LIN {X 0,Y 220.279,Z 449.432,A -85,B 0,C 180,E1 -22179.651,E2 -22179.651} C_VEL
LIN {X 0,Y 223.173,Z 455.881,A -85,B 0,C 180,E1 -22180.694,E2 -22180.694} C_VEL
LIN {X 0,Y 220.537,Z 499.361,A -85,B 0,C 180,E1 -22182.042,E2 -22182.042} C_VEL
LIN {X 0,Y 218.945,Z 512.319,A -85,B 0,C 180,E1 -22182.756,E2 -22182.756} C_VEL
LIN {X 0,Y 216.728,Z 525.067,A -85,B 0,C 180,E1 -22183.822,E2 -22183.822} C_VEL
LIN {X 0,Y 213.871,Z 536.29,A -85,B 0,C 180,E1 -22185.05,E2 -22185.05} C_VEL
LIN {X 0,Y 210.428,Z 547.967,A -85,B 0,C 180,E1 -22186.792,E2 -22186.792} C_VEL
LIN {X 0,Y 207.087,Z 557.88,A -85,B 0,C 180,E1 -22188.721,E2 -22188.721} C_VEL
LIN {X 0,Y 203.422,Z 566.935,A -85,B 0,C 180,E1 -22190.913,E2 -22190.913} C_VEL
LIN {X 0,Y 199.206,Z 576.115,A -85,B 0,C 180,E1 -22193.787,E2 -22193.787} C_VEL
LIN {X 0,Y 195.527,Z 583.431,A -85,B 0,C 180,E1 -22196.761,E2 -22196.761} C_VEL
LIN {X 0,Y 192.781,Z 588.357,A -85,B 0,C 180,E1 -22199.312,E2 -22199.312} C_VEL
LIN {X 0,Y 189.682,Z 593.549,A -85,B 0,C 180,E1 -22202.779,E2 -22202.779} C_VEL
LIN {X 0,Y 187.622,Z 596.712,A -85,B 0,C 180,E1 -22205.668,E2 -22205.668} C_VEL
LIN {X 0,Y 186.374,Z 598.548,A -85,B 0,C 180,E1 -22207.847,E2 -22207.847} C_VEL
LIN {X 0,Y 184.61,Z 600.806,A -85,B 0,C 180,E1 -22212.13,E2 -22212.13} C_VEL
LIN {X 0,Y 183.947,Z 601.411,A -85,B 0,C 180,E1 -22214.488,E2 -22214.488} C_VEL
LIN {X 0,Y 183.461,Z 601.557,A -85,B 0,C 180,E1 -22216.712,E2 -22216.712} C_VEL
LIN {X 0,Y 183.165,Z 600.608,A -85,B 0,C 180,E1 -22221.172,E2 -22221.172} C_VEL
LIN {X 0,Y 183.462,Z 598.591,A -85,B 0,C 180,E1 -22224.883,E2 -22224.883} C_VEL
LIN {X 0,Y 183.934,Z 595.067,A -85,B 0,C 180,E1 -22228.905,E2 -22228.905} C_VEL
LIN {X 0,Y 184.847,Z 591.015,A -85,B 0,C 180,E1 -22232.179,E2 -22232.179} C_VEL
LIN {X 0,Y 186.289,Z 584.814,A -85,B 0,C 180,E1 -22235.955,E2 -22235.955} C_VEL
LIN {X 0,Y 188.121,Z 578.059,A -85,B 0,C 180,E1 -22239.136,E2 -22239.136} C_VEL
LIN {X 0,Y 190.373,Z 569.662,A -85,B 0,C 180,E1 -22242.255,E2 -22242.255} C_VEL
LIN {X 0,Y 192.597,Z 561.018,A -85,B 0,C 180,E1 -22244.799,E2 -22244.799} C_VEL
LIN {X 0,Y 195.203,Z 550.369,A -85,B 0,C 180,E1 -22247.279,E2 -22247.279} C_VEL
LIN {X 0,Y 197.473,Z 539.775,A -85,B 0,C 180,E1 -22249.22,E2 -22249.22} C_VEL
LIN {X 0,Y 199.436,Z 527.973,A -85,B 0,C 180,E1 -22250.903,E2 -22250.903} C_VEL
LIN {X 0,Y 201.153,Z 515.679,A -85,B 0,C 180,E1 -22252.195,E2 -22252.195} C_VEL
LIN {X 0,Y 202.366,Z 502.967,A -85,B 0,C 180,E1 -22253.14,E2 -22253.14} C_VEL
LIN {X 0,Y 203.145,Z 489.487,A -85,B 0,C 180,E1 -22253.729,E2 -22253.729} C_VEL
LIN {X 0,Y 205.349,Z 437.648,A -85,B 0,C 180,E1 -22255.442,E2 -22255.442} C_VEL
LIN {X 0,Y 202.251,Z 429.977,A -85,B 0,C 180,E1 -22256.283,E2 -22256.283} C_VEL
LIN {X 0,Y 193.557,Z 412.703,A -85,B 0,C 180,E1 -22258.641,E2 -22258.641} C_VEL
LIN {X 0,Y 187.249,Z 402.11,A -85,B 0,C 180,E1 -22260.443,E2 -22260.443} C_VEL
LIN {X 0,Y 185.803,Z 399.476,A -85,B 0,C 180,E1 -22260.889,E2 -22260.889} C_VEL
LIN {X 0,Y 185.553,Z 398.371,A -85,B 0,C 180,E1 -22261.052,E2 -22261.052} C_VEL
LIN {X 0,Y 185.501,Z 398.377,A -85,B 0,C 180,E1 -22264.631,E2 -22264.631} C_VEL
LIN {X 0,Y 185.507,Z 398.376,A -85,B 0,C 180,E1 -22267.312,E2 -22267.312} C_VEL
LIN {X 0,Y 185.497,Z 398.375,A -85,B 0,C 180,E1 -22272.997,E2 -22272.997} C_VEL
LIN {X 0,Y 185.554,Z 398.352,A -85,B 0,C 180,E1 -22277.017,E2 -22277.017} C_VEL
LIN {X 0,Y 185.556,Z 398.366,A -85,B 0,C 180,E1 -22279.917,E2 -22279.917} C_VEL
LIN {X 0,Y 185.575,Z 398.362,A -85,B 0,C 180,E1 -22282.702,E2 -22282.702} C_VEL
LIN {X 0,Y 185.539,Z 398.368,A -85,B 0,C 180,E1 -22287.973,E2 -22287.973} C_VEL
LIN {X 0,Y 185.579,Z 398.367,A -85,B 0,C 180,E1 -22290.576,E2 -22290.576} C_VEL
LIN {X 0,Y 185.604,Z 398.344,A -85,B 0,C 180,E1 -22295.384,E2 -22295.384} C_VEL
LIN {X 0,Y 185.708,Z 398.347,A -85,B 0,C 180,E1 -22301.1,E2 -22301.1} C_VEL
LIN {X 0,Y 185.731,Z 398.337,A -85,B 0,C 180,E1 -22306.877,E2 -22306.877} C_VEL
LIN {X 0,Y 186.005,Z 398.311,A -85,B 0,C 180,E1 -22311.307,E2 -22311.307} C_VEL
LIN {X 0,Y 186.203,Z 398.28,A -85,B 0,C 180,E1 -22317.836,E2 -22317.836} C_VEL
LIN {X 0,Y 186.405,Z 398.265,A -85,B 0,C 180,E1 -22319.999,E2 -22319.999} C_VEL
LIN {X 0,Y 185.922,Z 398.322,A -85,B 0,C 180,E1 -22324.335,E2 -22324.335} C_VEL
LIN {X 0,Y 186.005,Z 398.309,A -85,B 0,C 180,E1 -22328.692,E2 -22328.692} C_VEL
LIN {X 0,Y 185.76,Z 398.341,A -85,B 0,C 180,E1 -22333.12,E2 -22333.12} C_VEL
LIN {X 0,Y 185.713,Z 398.35,A -85,B 0,C 180,E1 -22337.622,E2 -22337.622} C_VEL
LIN {X 0,Y 185.612,Z 398.363,A -85,B 0,C 180,E1 -22342.249,E2 -22342.249} C_VEL
LIN {X 0,Y 185.558,Z 398.371,A -85,B 0,C 180,E1 -22347.032,E2 -22347.032} C_VEL
LIN {X 0,Y 185.574,Z 398.369,A -85,B 0,C 180,E1 -22349.493,E2 -22349.493} C_VEL
LIN {X 0,Y 185.517,Z 398.377,A -85,B 0,C 180,E1 -22354.628,E2 -22354.628} C_VEL
LIN {X 0,Y 185.565,Z 398.371,A -85,B 0,C 180,E1 -22357.314,E2 -22357.314} C_VEL
LIN {X 0,Y 185.559,Z 398.372,A -85,B 0,C 180,E1 -22360.758,E2 -22360.758} C_VEL
LIN {X 0,Y 185.555,Z 398.372,A -85,B 0,C 180,E1 -22363.977,E2 -22363.977} C_VEL
LIN {X 0,Y 185.528,Z 398.445,A -85,B 0,C 180,E1 -22366.131,E2 -22366.131} C_VEL
LIN {X 0,Y 187.321,Z 405.414,A -85,B 0,C 180,E1 -22370.086,E2 -22370.086} C_VEL
LIN {X 0,Y 193.699,Z 418.874,A -85,B 0,C 180,E1 -22372.016,E2 -22372.016} C_VEL
LIN {X 0,Y 199.309,Z 432.552,A -85,B 0,C 180,E1 -22373.66,E2 -22373.66} C_VEL
LIN {X 0,Y 201.553,Z 438.763,A -85,B 0,C 180,E1 -22374.315,E2 -22374.315} C_VEL
LIN {X 0,Y 204.313,Z 466.927,A -85,B 0,C 180,E1 -22375.916,E2 -22375.916} C_VEL
LIN {X 0,Y 203.519,Z 486.913,A -85,B 0,C 180,E1 -22376.586,E2 -22376.586} C_VEL
LIN {X 0,Y 202.708,Z 492.757,A -85,B 0,C 180,E1 -22376.683,E2 -22376.683} C_VEL
LIN {X 0,Y 197.313,Z 509.789,A -85,B 0,C 180,E1 -22376.528,E2 -22376.528} C_VEL
LIN {X 0,Y 195.967,Z 515.551,A -85,B 0,C 180,E1 -22376.62,E2 -22376.62} C_VEL
LIN {X 0,Y 195.732,Z 517.491,A -85,B 0,C 180,E1 -22376.71,E2 -22376.71} C_VEL
LIN {X 0,Y 194.346,Z 530.518,A -85,B 0,C 180,E1 -22377.613,E2 -22377.613} C_VEL
LIN {X 0,Y 192.342,Z 543.335,A -85,B 0,C 180,E1 -22378.929,E2 -22378.929} C_VEL
LIN {X 0,Y 190.213,Z 553.96,A -85,B 0,C 180,E1 -22380.385,E2 -22380.385} C_VEL
LIN {X 0,Y 187.569,Z 565.212,A -85,B 0,C 180,E1 -22382.376,E2 -22382.376} C_VEL
LIN {X 0,Y 185.007,Z 575.331,A -85,B 0,C 180,E1 -22384.7,E2 -22384.7} C_VEL
LIN {X 0,Y 182.55,Z 584.487,A -85,B 0,C 180,E1 -22387.357,E2 -22387.357} C_VEL
LIN {X 0,Y 180.701,Z 592.065,A -85,B 0,C 180,E1 -22390.105,E2 -22390.105} C_VEL
LIN {X 0,Y 178.739,Z 599.477,A -85,B 0,C 180,E1 -22393.437,E2 -22393.437} C_VEL
LIN {X 0,Y 177.463,Z 604.489,A -85,B 0,C 180,E1 -22396.254,E2 -22396.254} C_VEL
LIN {X 0,Y 176.631,Z 609.363,A -85,B 0,C 180,E1 -22399.686,E2 -22399.686} C_VEL
LIN {X 0,Y 176.218,Z 613.088,A -85,B 0,C 180,E1 -22403.128,E2 -22403.128} C_VEL
LIN {X 0,Y 176.155,Z 615.331,A -85,B 0,C 180,E1 -22405.878,E2 -22405.878} C_VEL
LIN {X 0,Y 176.349,Z 617.484,A -85,B 0,C 180,E1 -22410,E2 -22410} C_VEL
LIN {X 0,Y 176.071,Z 618.254,A -85,B 0,C 180,E1 -22413.723,E2 -22413.723} C_VEL
LIN {X 0,Y 176.128,Z 618.102,A -85,B 0,C 180,E1 -22416.875,E2 -22416.875} C_VEL
LIN {X 0,Y 176.942,Z 616.5,A -85,B 0,C 180,E1 -22421.455,E2 -22421.455} C_VEL
LIN {X 0,Y 177.674,Z 615.118,A -85,B 0,C 180,E1 -22423.729,E2 -22423.729} C_VEL
LIN {X 0,Y 179.338,Z 612.237,A -85,B 0,C 180,E1 -22427.092,E2 -22427.092} C_VEL
LIN {X 0,Y 181.645,Z 608.353,A -85,B 0,C 180,E1 -22430.378,E2 -22430.378} C_VEL
LIN {X 0,Y 184.564,Z 603.367,A -85,B 0,C 180,E1 -22433.567,E2 -22433.567} C_VEL
LIN {X 0,Y 187.821,Z 597.127,A -85,B 0,C 180,E1 -22436.68,E2 -22436.68} C_VEL
LIN {X 0,Y 191.864,Z 589.376,A -85,B 0,C 180,E1 -22439.636,E2 -22439.636} C_VEL
LIN {X 0,Y 196.489,Z 579.698,A -85,B 0,C 180,E1 -22442.446,E2 -22442.446} C_VEL
LIN {X 0,Y 200.738,Z 569.726,A -85,B 0,C 180,E1 -22444.674,E2 -22444.674} C_VEL
LIN {X 0,Y 204.817,Z 558.474,A -85,B 0,C 180,E1 -22446.597,E2 -22446.597} C_VEL
LIN {X 0,Y 208.195,Z 547.47,A -85,B 0,C 180,E1 -22448.028,E2 -22448.028} C_VEL
LIN {X 0,Y 211.236,Z 535.284,A -85,B 0,C 180,E1 -22449.208,E2 -22449.208} C_VEL
LIN {X 0,Y 213.545,Z 522.568,A -85,B 0,C 180,E1 -22450.072,E2 -22450.072} C_VEL
LIN {X 0,Y 215.104,Z 508.485,A -85,B 0,C 180,E1 -22450.679,E2 -22450.679} C_VEL
LIN {X 0,Y 217.075,Z 473.858,A -85,B 0,C 180,E1 -22451.765,E2 -22451.765} C_VEL
LIN {X 0,Y 216.264,Z 466.923,A -85,B 0,C 180,E1 -22452.308,E2 -22452.308} C_VEL
LIN {X 0,Y 211.577,Z 455.568,A -85,B 0,C 180,E1 -22454.198,E2 -22454.198} C_VEL
LIN {X 0,Y 206.02,Z 443.944,A -85,B 0,C 180,E1 -22456.558,E2 -22456.558} C_VEL
LIN {X 0,Y 201.04,Z 434.777,A -85,B 0,C 180,E1 -22458.824,E2 -22458.824} C_VEL
LIN {X 0,Y 197.955,Z 429.38,A -85,B 0,C 180,E1 -22460.335,E2 -22460.335} C_VEL
LIN {X 0,Y 195.318,Z 425.091,A -85,B 0,C 180,E1 -22461.691,E2 -22461.691} C_VEL
LIN {X 0,Y 192.281,Z 420.183,A -85,B 0,C 180,E1 -22463.36,E2 -22463.36} C_VEL
LIN {X 0,Y 189.015,Z 415.191,A -85,B 0,C 180,E1 -22465.29,E2 -22465.29} C_VEL
LIN {X 0,Y 185.075,Z 409.818,A -85,B 0,C 180,E1 -22467.827,E2 -22467.827} C_VEL
LIN {X 0,Y 183.945,Z 408.105,A -85,B 0,C 180,E1 -22468.63,E2 -22468.63} C_VEL
LIN {X 0,Y 180.436,Z 403.71,A -85,B 0,C 180,E1 -22471.262,E2 -22471.262} C_VEL
LIN {X 0,Y 179.325,Z 401.668,A -85,B 0,C 180,E1 -22472.264,E2 -22472.264} C_VEL
LIN {X 0,Y 178.541,Z 399.205,A -85,B 0,C 180,E1 -22475.475,E2 -22475.475} C_VEL
LIN {X 0,Y 178.646,Z 399.223,A -85,B 0,C 180,E1 -22481.656,E2 -22481.656} C_VEL
LIN {X 0,Y 178.677,Z 399.222,A -85,B 0,C 180,E1 -22486.35,E2 -22486.35} C_VEL
LIN {X 0,Y 178.959,Z 399.187,A -85,B 0,C 180,E1 -22490.963,E2 -22490.963} C_VEL
LIN {X 0,Y 179.15,Z 399.16,A -85,B 0,C 180,E1 -22497.752,E2 -22497.752} C_VEL
LIN {X 0,Y 179.368,Z 399.134,A -85,B 0,C 180,E1 -22500.001,E2 -22500.001} C_VEL
LIN {X 0,Y 178.863,Z 399.195,A -85,B 0,C 180,E1 -22504.508,E2 -22504.508} C_VEL
LIN {X 0,Y 178.908,Z 399.189,A -85,B 0,C 180,E1 -22509.041,E2 -22509.041} C_VEL
LIN {X 0,Y 178.654,Z 399.222,A -85,B 0,C 180,E1 -22513.653,E2 -22513.653} C_VEL
LIN {X 0,Y 178.656,Z 399.24,A -85,B 0,C 180,E1 -22518.714,E2 -22518.714} C_VEL
LIN {X 0,Y 179.292,Z 401.493,A -85,B 0,C 180,E1 -22519.406,E2 -22519.406} C_VEL
LIN {X 0,Y 180.93,Z 403.727,A -85,B 0,C 180,E1 -22520.76,E2 -22520.76} C_VEL
LIN {X 0,Y 183.354,Z 405.343,A -85,B 0,C 180,E1 -22522.465,E2 -22522.465} C_VEL
LIN {X 0,Y 185.051,Z 408.386,A -85,B 0,C 180,E1 -22523.73,E2 -22523.73} C_VEL
LIN {X 0,Y 187.649,Z 410.827,A -85,B 0,C 180,E1 -22525.364,E2 -22525.364} C_VEL
LIN {X 0,Y 189.966,Z 414.17,A -85,B 0,C 180,E1 -22526.802,E2 -22526.802} C_VEL
LIN {X 0,Y 191.627,Z 415.94,A -85,B 0,C 180,E1 -22527.732,E2 -22527.732} C_VEL
LIN {X 0,Y 194.227,Z 419.503,A -85,B 0,C 180,E1 -22529.161,E2 -22529.161} C_VEL
LIN {X 0,Y 198.844,Z 425.908,A -85,B 0,C 180,E1 -22531.496,E2 -22531.496} C_VEL
LIN {X 0,Y 203.808,Z 432.939,A -85,B 0,C 180,E1 -22533.766,E2 -22533.766} C_VEL
LIN {X 0,Y 210.132,Z 443.126,A -85,B 0,C 180,E1 -22536.418,E2 -22536.418} C_VEL
LIN {X 0,Y 216.149,Z 454.069,A -85,B 0,C 180,E1 -22538.741,E2 -22538.741} C_VEL
LIN {X 0,Y 218.063,Z 458.718,A -85,B 0,C 180,E1 -22539.486,E2 -22539.486} C_VEL
LIN {X 0,Y 215.395,Z 499.783,A -85,B 0,C 180,E1 -22540.763,E2 -22540.763} C_VEL
LIN {X 0,Y 213.731,Z 512.785,A -85,B 0,C 180,E1 -22541.489,E2 -22541.489} C_VEL
LIN {X 0,Y 211.541,Z 524.945,A -85,B 0,C 180,E1 -22542.514,E2 -22542.514} C_VEL
LIN {X 0,Y 208.345,Z 537.095,A -85,B 0,C 180,E1 -22543.862,E2 -22543.862} C_VEL
LIN {X 0,Y 204.765,Z 548.685,A -85,B 0,C 180,E1 -22545.629,E2 -22545.629} C_VEL
LIN {X 0,Y 201.511,Z 557.933,A -85,B 0,C 180,E1 -22547.465,E2 -22547.465} C_VEL
LIN {X 0,Y 197.84,Z 566.65,A -85,B 0,C 180,E1 -22549.587,E2 -22549.587} C_VEL
LIN {X 0,Y 194.113,Z 574.567,A -85,B 0,C 180,E1 -22552.013,E2 -22552.013} C_VEL
LIN {X 0,Y 190.109,Z 582.242,A -85,B 0,C 180,E1 -22555.041,E2 -22555.041} C_VEL
LIN {X 0,Y 186.559,Z 588.37,A -85,B 0,C 180,E1 -22558.171,E2 -22558.171} C_VEL
LIN {X 0,Y 183.49,Z 593.262,A -85,B 0,C 180,E1 -22561.457,E2 -22561.457} C_VEL
LIN {X 0,Y 181.018,Z 596.859,A -85,B 0,C 180,E1 -22564.719,E2 -22564.719} C_VEL
LIN {X 0,Y 179.672,Z 598.736,A -85,B 0,C 180,E1 -22566.974,E2 -22566.974} C_VEL
LIN {X 0,Y 178.572,Z 600.14,A -85,B 0,C 180,E1 -22569.256,E2 -22569.256} C_VEL
LIN {X 0,Y 177.622,Z 601.181,A -85,B 0,C 180,E1 -22571.737,E2 -22571.737} C_VEL
LIN {X 0,Y 176.47,Z 601.902,A -85,B 0,C 180,E1 -22576.176,E2 -22576.176} C_VEL
LIN {X 0,Y 176.161,Z 601.657,A -85,B 0,C 180,E1 -22578.494,E2 -22578.494} C_VEL
LIN {X 0,Y 176.186,Z 599.991,A -85,B 0,C 180,E1 -22583.127,E2 -22583.127} C_VEL
LIN {X 0,Y 176.399,Z 598.563,A -85,B 0,C 180,E1 -22585.43,E2 -22585.43} C_VEL
LIN {X 0,Y 176.841,Z 595.613,A -85,B 0,C 180,E1 -22588.861,E2 -22588.861} C_VEL
LIN {X 0,Y 177.757,Z 591.626,A -85,B 0,C 180,E1 -22592.266,E2 -22592.266} C_VEL
LIN {X 0,Y 179.259,Z 585.506,A -85,B 0,C 180,E1 -22596.189,E2 -22596.189} C_VEL
LIN {X 0,Y 181.119,Z 578.835,A -85,B 0,C 180,E1 -22599.492,E2 -22599.492} C_VEL
LIN {X 0,Y 183.462,Z 570.561,A -85,B 0,C 180,E1 -22602.725,E2 -22602.725} C_VEL
LIN {X 0,Y 185.771,Z 562.049,A -85,B 0,C 180,E1 -22605.356,E2 -22605.356} C_VEL
LIN {X 0,Y 188.487,Z 551.537,A -85,B 0,C 180,E1 -22607.915,E2 -22607.915} C_VEL
LIN {X 0,Y 190.829,Z 541.127,A -85,B 0,C 180,E1 -22609.917,E2 -22609.917} C_VEL
LIN {X 0,Y 192.877,Z 529.709,A -85,B 0,C 180,E1 -22611.649,E2 -22611.649} C_VEL
LIN {X 0,Y 194.833,Z 516.562,A -85,B 0,C 180,E1 -22613.096,E2 -22613.096} C_VEL
LIN {X 0,Y 196.131,Z 503.702,A -85,B 0,C 180,E1 -22614.091,E2 -22614.091} C_VEL
LIN {X 0,Y 196.916,Z 490.753,A -85,B 0,C 180,E1 -22614.692,E2 -22614.692} C_VEL
LIN {X 0,Y 199.231,Z 439.293,A -85,B 0,C 180,E1 -22616.431,E2 -22616.431} C_VEL
LIN {X 0,Y 194.308,Z 428.224,A -85,B 0,C 180,E1 -22617.815,E2 -22617.815} C_VEL
LIN {X 0,Y 186.993,Z 414.064,A -85,B 0,C 180,E1 -22619.945,E2 -22619.945} C_VEL
LIN {X 0,Y 180.425,Z 403.251,A -85,B 0,C 180,E1 -22621.964,E2 -22621.964} C_VEL
LIN {X 0,Y 178.822,Z 400.699,A -85,B 0,C 180,E1 -22622.484,E2 -22622.484} C_VEL
LIN {X 0,Y 178.497,Z 399.25,A -85,B 0,C 180,E1 -22622.686,E2 -22622.686} C_VEL
LIN {X 0,Y 178.439,Z 399.258,A -85,B 0,C 180,E1 -22628.026,E2 -22628.026} C_VEL
LIN {X 0,Y 178.419,Z 399.249,A -85,B 0,C 180,E1 -22632.038,E2 -22632.038} C_VEL
LIN {X 0,Y 178.462,Z 399.25,A -85,B 0,C 180,E1 -22635.141,E2 -22635.141} C_VEL
LIN {X 0,Y 178.506,Z 399.232,A -85,B 0,C 180,E1 -22638.421,E2 -22638.421} C_VEL
LIN {X 0,Y 178.467,Z 399.237,A -85,B 0,C 180,E1 -22643.792,E2 -22643.792} C_VEL
LIN {X 0,Y 178.488,Z 399.232,A -85,B 0,C 180,E1 -22646.546,E2 -22646.546} C_VEL
LIN {X 0,Y 178.52,Z 399.249,A -85,B 0,C 180,E1 -22650.006,E2 -22650.006} C_VEL
LIN {X 0,Y 178.533,Z 399.221,A -85,B 0,C 180,E1 -22654.875,E2 -22654.875} C_VEL
LIN {X 0,Y 178.652,Z 399.227,A -85,B 0,C 180,E1 -22660.754,E2 -22660.754} C_VEL
LIN {X 0,Y 178.658,Z 399.212,A -85,B 0,C 180,E1 -22666.347,E2 -22666.347} C_VEL
LIN {X 0,Y 178.956,Z 399.189,A -85,B 0,C 180,E1 -22670.961,E2 -22670.961} C_VEL
LIN {X 0,Y 179.149,Z 399.157,A -85,B 0,C 180,E1 -22677.751,E2 -22677.751} C_VEL
LIN {X 0,Y 179.368,Z 399.141,A -85,B 0,C 180,E1 -22679.999,E2 -22679.999} C_VEL
LIN {X 0,Y 178.87,Z 399.202,A -85,B 0,C 180,E1 -22684.507,E2 -22684.507} C_VEL
LIN {X 0,Y 178.956,Z 399.188,A -85,B 0,C 180,E1 -22689.037,E2 -22689.037} C_VEL
LIN {X 0,Y 178.683,Z 399.221,A -85,B 0,C 180,E1 -22693.65,E2 -22693.65} C_VEL
LIN {X 0,Y 178.676,Z 399.222,A -85,B 0,C 180,E1 -22698.34,E2 -22698.34} C_VEL
LIN {X 0,Y 178.526,Z 399.243,A -85,B 0,C 180,E1 -22703.182,E2 -22703.182} C_VEL
LIN {X 0,Y 178.483,Z 399.249,A -85,B 0,C 180,E1 -22708.197,E2 -22708.197} C_VEL
LIN {X 0,Y 178.474,Z 399.255,A -85,B 0,C 180,E1 -22710.791,E2 -22710.791} C_VEL
LIN {X 0,Y 178.481,Z 399.255,A -85,B 0,C 180,E1 -22714.219,E2 -22714.219} C_VEL
LIN {X 0,Y 178.47,Z 399.255,A -85,B 0,C 180,E1 -22719.055,E2 -22719.055} C_VEL
LIN {X 0,Y 178.496,Z 399.248,A -85,B 0,C 180,E1 -22722.016,E2 -22722.016} C_VEL
LIN {X 0,Y 178.488,Z 399.421,A -85,B 0,C 180,E1 -22725.018,E2 -22725.018} C_VEL
LIN {X 0,Y 179.966,Z 405.005,A -85,B 0,C 180,E1 -22728.371,E2 -22728.371} C_VEL
LIN {X 0,Y 182.169,Z 409.272,A -85,B 0,C 180,E1 -22729.104,E2 -22729.104} C_VEL
LIN {X 0,Y 188.362,Z 422.421,A -85,B 0,C 180,E1 -22731.09,E2 -22731.09} C_VEL
LIN {X 0,Y 193.401,Z 434.627,A -85,B 0,C 180,E1 -22732.647,E2 -22732.647} C_VEL
LIN {X 0,Y 195.655,Z 440.931,A -85,B 0,C 180,E1 -22733.345,E2 -22733.345} C_VEL
LIN {X 0,Y 198.181,Z 468.607,A -85,B 0,C 180,E1 -22734.963,E2 -22734.963} C_VEL
LIN {X 0,Y 195.995,Z 514.323,A -85,B 0,C 180,E1 -22736.548,E2 -22736.548} C_VEL
LIN {X 0,Y 195.732,Z 517.491,A -85,B 0,C 180,E1 -22736.71,E2 -22736.71} C_VEL
LIN {X 0,Y 194.561,Z 523.244,A -85,B 0,C 180,E1 -22736.943,E2 -22736.943} C_VEL
LIN {X 0,Y 190.887,Z 532.419,A -85,B 0,C 180,E1 -22737.251,E2 -22737.251} C_VEL
LIN {X 0,Y 186.915,Z 541.333,A -85,B 0,C 180,E1 -22737.792,E2 -22737.792} C_VEL
LIN {X 0,Y 185.293,Z 546.671,A -85,B 0,C 180,E1 -22738.394,E2 -22738.394} C_VEL
LIN {X 0,Y 182.646,Z 558.79,A -85,B 0,C 180,E1 -22740.304,E2 -22740.304} C_VEL
LIN {X 0,Y 180.09,Z 569.014,A -85,B 0,C 180,E1 -22742.393,E2 -22742.393} C_VEL
LIN {X 0,Y 177.464,Z 578.393,A -85,B 0,C 180,E1 -22744.804,E2 -22744.804} C_VEL
LIN {X 0,Y 174.896,Z 587.403,A -85,B 0,C 180,E1 -22747.749,E2 -22747.749} C_VEL
LIN {X 0,Y 173.575,Z 592.726,A -85,B 0,C 180,E1 -22749.87,E2 -22749.87} C_VEL
LIN {X 0,Y 171.611,Z 599.955,A -85,B 0,C 180,E1 -22753.342,E2 -22753.342} C_VEL
LIN {X 0,Y 170.166,Z 605.701,A -85,B 0,C 180,E1 -22756.871,E2 -22756.871} C_VEL
LIN {X 0,Y 169.395,Z 610.227,A -85,B 0,C 180,E1 -22760.448,E2 -22760.448} C_VEL
LIN {X 0,Y 169.146,Z 612.609,A -85,B 0,C 180,E1 -22762.84,E2 -22762.84} C_VEL
LIN {X 0,Y 169.074,Z 615.105,A -85,B 0,C 180,E1 -22766.042,E2 -22766.042} C_VEL
LIN {X 0,Y 169.266,Z 617.097,A -85,B 0,C 180,E1 -22770,E2 -22770} C_VEL
LIN {X 0,Y 169.011,Z 617.898,A -85,B 0,C 180,E1 -22773.635,E2 -22773.635} C_VEL
LIN {X 0,Y 169.078,Z 617.795,A -85,B 0,C 180,E1 -22777.163,E2 -22777.163} C_VEL
LIN {X 0,Y 169.969,Z 616.242,A -85,B 0,C 180,E1 -22781.931,E2 -22781.931} C_VEL
LIN {X 0,Y 171.831,Z 613.123,A -85,B 0,C 180,E1 -22786.636,E2 -22786.636} C_VEL
LIN {X 0,Y 174.148,Z 609.634,A -85,B 0,C 180,E1 -22790.061,E2 -22790.061} C_VEL
LIN {X 0,Y 177.661,Z 603.959,A -85,B 0,C 180,E1 -22794.08,E2 -22794.08} C_VEL
LIN {X 0,Y 181.501,Z 597.101,A -85,B 0,C 180,E1 -22797.687,E2 -22797.687} C_VEL
LIN {X 0,Y 185.716,Z 589.447,A -85,B 0,C 180,E1 -22800.721,E2 -22800.721} C_VEL
LIN {X 0,Y 190.541,Z 579.857,A -85,B 0,C 180,E1 -22803.59,E2 -22803.59} C_VEL
LIN {X 0,Y 194.941,Z 569.987,A -85,B 0,C 180,E1 -22805.862,E2 -22805.862} C_VEL
LIN {X 0,Y 199.181,Z 558.929,A -85,B 0,C 180,E1 -22807.811,E2 -22807.811} C_VEL
LIN {X 0,Y 202.681,Z 548.113,A -85,B 0,C 180,E1 -22809.257,E2 -22809.257} C_VEL
LIN {X 0,Y 205.818,Z 536.198,A -85,B 0,C 180,E1 -22810.449,E2 -22810.449} C_VEL
LIN {X 0,Y 208.386,Z 523.059,A -85,B 0,C 180,E1 -22811.382,E2 -22811.382} C_VEL
LIN {X 0,Y 210.024,Z 509.109,A -85,B 0,C 180,E1 -22812.008,E2 -22812.008} C_VEL
LIN {X 0,Y 212.097,Z 474.746,A -85,B 0,C 180,E1 -22813.102,E2 -22813.102} C_VEL
LIN {X 0,Y 211.483,Z 469.879,A -85,B 0,C 180,E1 -22813.518,E2 -22813.518} C_VEL
LIN {X 0,Y 206.811,Z 458.449,A -85,B 0,C 180,E1 -22815.53,E2 -22815.53} C_VEL
LIN {X 0,Y 201.814,Z 447.81,A -85,B 0,C 180,E1 -22817.799,E2 -22817.799} C_VEL
LIN {X 0,Y 196.83,Z 438.474,A -85,B 0,C 180,E1 -22820.231,E2 -22820.231} C_VEL
LIN {X 0,Y 192.412,Z 430.785,A -85,B 0,C 180,E1 -22822.591,E2 -22822.591} C_VEL
LIN {X 0,Y 189.315,Z 425.776,A -85,B 0,C 180,E1 -22824.38,E2 -22824.38} C_VEL
LIN {X 0,Y 185.745,Z 420.294,A -85,B 0,C 180,E1 -22826.626,E2 -22826.626} C_VEL
LIN {X 0,Y 182.125,Z 414.805,A -85,B 0,C 180,E1 -22829.174,E2 -22829.174} C_VEL
LIN {X 0,Y 178.314,Z 409.867,A -85,B 0,C 180,E1 -22832.173,E2 -22832.173} C_VEL
LIN {X 0,Y 177.207,Z 408.001,A -85,B 0,C 180,E1 -22833.184,E2 -22833.184} C_VEL
LIN {X 0,Y 174.048,Z 404.686,A -85,B 0,C 180,E1 -22836.185,E2 -22836.185} C_VEL
LIN {X 0,Y 172.237,Z 402.566,A -85,B 0,C 180,E1 -22838.219,E2 -22838.219} C_VEL
LIN {X 0,Y 171.571,Z 400.618,A -85,B 0,C 180,E1 -22839.254,E2 -22839.254} C_VEL
LIN {X 0,Y 171.541,Z 400.106,A -85,B 0,C 180,E1 -22840.439,E2 -22840.439} C_VEL
LIN {X 0,Y 171.589,Z 400.1,A -85,B 0,C 180,E1 -22845.774,E2 -22845.774} C_VEL
LIN {X 0,Y 171.888,Z 400.065,A -85,B 0,C 180,E1 -22850.588,E2 -22850.588} C_VEL
LIN {X 0,Y 171.82,Z 400.073,A -85,B 0,C 180,E1 -22855.308,E2 -22855.308} C_VEL
LIN {X 0,Y 172.331,Z 400.01,A -85,B 0,C 180,E1 -22860.001,E2 -22860.001} C_VEL
LIN {X 0,Y 171.812,Z 400.074,A -85,B 0,C 180,E1 -22864.693,E2 -22864.693} C_VEL
LIN {X 0,Y 171.845,Z 400.071,A -85,B 0,C 180,E1 -22869.416,E2 -22869.416} C_VEL
LIN {X 0,Y 171.639,Z 400.124,A -85,B 0,C 180,E1 -22872.489,E2 -22872.489} C_VEL
LIN {X 0,Y 172.34,Z 402.449,A -85,B 0,C 180,E1 -22873.562,E2 -22873.562} C_VEL
LIN {X 0,Y 174.06,Z 404.678,A -85,B 0,C 180,E1 -22875.516,E2 -22875.516} C_VEL
LIN {X 0,Y 176.644,Z 406.279,A -85,B 0,C 180,E1 -22877.885,E2 -22877.885} C_VEL
LIN {X 0,Y 178.116,Z 409.144,A -85,B 0,C 180,E1 -22879.296,E2 -22879.296} C_VEL
LIN {X 0,Y 180.437,Z 411.297,A -85,B 0,C 180,E1 -22881.119,E2 -22881.119} C_VEL
LIN {X 0,Y 181.225,Z 411.951,A -85,B 0,C 180,E1 -22881.693,E2 -22881.693} C_VEL
LIN {X 0,Y 183.498,Z 415.393,A -85,B 0,C 180,E1 -22883.391,E2 -22883.391} C_VEL
LIN {X 0,Y 185.323,Z 417.144,A -85,B 0,C 180,E1 -22884.581,E2 -22884.581} C_VEL
LIN {X 0,Y 187.886,Z 420.686,A -85,B 0,C 180,E1 -22886.223,E2 -22886.223} C_VEL
LIN {X 0,Y 189.296,Z 422.453,A -85,B 0,C 180,E1 -22887.063,E2 -22887.063} C_VEL
LIN {X 0,Y 193.189,Z 427.868,A -85,B 0,C 180,E1 -22889.251,E2 -22889.251} C_VEL
LIN {X 0,Y 198.271,Z 435.055,A -85,B 0,C 180,E1 -22891.822,E2 -22891.822} C_VEL
LIN {X 0,Y 204.792,Z 445.291,A -85,B 0,C 180,E1 -22894.788,E2 -22894.788} C_VEL
LIN {X 0,Y 211.752,Z 457.934,A -85,B 0,C 180,E1 -22897.659,E2 -22897.659} C_VEL
LIN {X 0,Y 213.027,Z 460.836,A -85,B 0,C 180,E1 -22898.177,E2 -22898.177} C_VEL
LIN {X 0,Y 210.356,Z 500.265,A -85,B 0,C 180,E1 -22899.423,E2 -22899.423} C_VEL
LIN {X 0,Y 208.62,Z 513.248,A -85,B 0,C 180,E1 -22900.157,E2 -22900.157} C_VEL
LIN {X 0,Y 206.233,Z 525.919,A -85,B 0,C 180,E1 -22901.251,E2 -22901.251} C_VEL
LIN {X 0,Y 202.909,Z 537.9,A -85,B 0,C 180,E1 -22902.608,E2 -22902.608} C_VEL
LIN {X 0,Y 199.201,Z 549.404,A -85,B 0,C 180,E1 -22904.404,E2 -22904.404} C_VEL
LIN {X 0,Y 195.464,Z 559.395,A -85,B 0,C 180,E1 -22906.448,E2 -22906.448} C_VEL
LIN {X 0,Y 191.561,Z 568.089,A -85,B 0,C 180,E1 -22908.672,E2 -22908.672} C_VEL
LIN {X 0,Y 187.699,Z 575.794,A -85,B 0,C 180,E1 -22911.16,E2 -22911.16} C_VEL
LIN {X 0,Y 183.522,Z 583.358,A -85,B 0,C 180,E1 -22914.3,E2 -22914.3} C_VEL
LIN {X 0,Y 179.302,Z 590.172,A -85,B 0,C 180,E1 -22918.053,E2 -22918.053} C_VEL
LIN {X 0,Y 176.236,Z 594.656,A -85,B 0,C 180,E1 -22921.411,E2 -22921.411} C_VEL
LIN {X 0,Y 174.484,Z 597.007,A -85,B 0,C 180,E1 -22923.701,E2 -22923.701} C_VEL
LIN {X 0,Y 173.003,Z 598.916,A -85,B 0,C 180,E1 -22926.032,E2 -22926.032} C_VEL
LIN {X 0,Y 171.811,Z 600.379,A -85,B 0,C 180,E1 -22928.399,E2 -22928.399} C_VEL
LIN {X 0,Y 170.054,Z 602.003,A -85,B 0,C 180,E1 -22933.185,E2 -22933.185} C_VEL
LIN {X 0,Y 169.497,Z 602.23,A -85,B 0,C 180,E1 -22935.595,E2 -22935.595} C_VEL
LIN {X 0,Y 169.107,Z 602.039,A -85,B 0,C 180,E1 -22938.007,E2 -22938.007} C_VEL
LIN {X 0,Y 169.082,Z 600.427,A -85,B 0,C 180,E1 -22942.837,E2 -22942.837} C_VEL
LIN {X 0,Y 169.299,Z 599.039,A -85,B 0,C 180,E1 -22945.238,E2 -22945.238} C_VEL
LIN {X 0,Y 169.751,Z 596.139,A -85,B 0,C 180,E1 -22948.814,E2 -22948.814} C_VEL
LIN {X 0,Y 170.65,Z 592.216,A -85,B 0,C 180,E1 -22952.36,E2 -22952.36} C_VEL
LIN {X 0,Y 171.965,Z 587.173,A -85,B 0,C 180,E1 -22955.864,E2 -22955.864} C_VEL
LIN {X 0,Y 173.772,Z 580.83,A -85,B 0,C 180,E1 -22959.31,E2 -22959.31} C_VEL
LIN {X 0,Y 176.127,Z 572.899,A -85,B 0,C 180,E1 -22962.677,E2 -22962.677} C_VEL
LIN {X 0,Y 178.966,Z 563.047,A -85,B 0,C 180,E1 -22965.955,E2 -22965.955} C_VEL
LIN {X 0,Y 181.769,Z 552.696,A -85,B 0,C 180,E1 -22968.601,E2 -22968.601} C_VEL
LIN {X 0,Y 184.518,Z 541.044,A -85,B 0,C 180,E1 -22970.92,E2 -22970.92} C_VEL
LIN {X 0,Y 186.689,Z 529.465,A -85,B 0,C 180,E1 -22972.697,E2 -22972.697} C_VEL
LIN {X 0,Y 188.547,Z 517.427,A -85,B 0,C 180,E1 -22974.059,E2 -22974.059} C_VEL
LIN {X 0,Y 189.962,Z 504.222,A -85,B 0,C 180,E1 -22975.117,E2 -22975.117} C_VEL
LIN {X 0,Y 190.756,Z 491.853,A -85,B 0,C 180,E1 -22975.721,E2 -22975.721} C_VEL
LIN {X 0,Y 193.167,Z 441.045,A -85,B 0,C 180,E1 -22977.477,E2 -22977.477} C_VEL
LIN {X 0,Y 186.81,Z 427.392,A -85,B 0,C 180,E1 -22979.37,E2 -22979.37} C_VEL
LIN {X 0,Y 180.268,Z 415.235,A -85,B 0,C 180,E1 -22981.414,E2 -22981.414} C_VEL
LIN {X 0,Y 173.369,Z 404.15,A -85,B 0,C 180,E1 -22983.713,E2 -22983.713} C_VEL
LIN {X 0,Y 171.848,Z 401.715,A -85,B 0,C 180,E1 -22984.253,E2 -22984.253} C_VEL
LIN {X 0,Y 171.434,Z 400.129,A -85,B 0,C 180,E1 -22984.473,E2 -22984.473} C_VEL
LIN {X 0,Y 171.361,Z 400.138,A -85,B 0,C 180,E1 -22988.807,E2 -22988.807} C_VEL
LIN {X 0,Y 171.368,Z 400.138,A -85,B 0,C 180,E1 -22994.201,E2 -22994.201} C_VEL
LIN {X 0,Y 171.424,Z 400.118,A -85,B 0,C 180,E1 -22999.006,E2 -22999.006} C_VEL
LIN {X 0,Y 171.44,Z 400.126,A -85,B 0,C 180,E1 -23002.054,E2 -23002.054} C_VEL
LIN {X 0,Y 171.417,Z 400.126,A -85,B 0,C 180,E1 -23007.791,E2 -23007.791} C_VEL
LIN {X 0,Y 171.446,Z 400.127,A -85,B 0,C 180,E1 -23010.533,E2 -23010.533} C_VEL
LIN {X 0,Y 171.464,Z 400.107,A -85,B 0,C 180,E1 -23015.802,E2 -23015.802} C_VEL
LIN {X 0,Y 171.608,Z 400.104,A -85,B 0,C 180,E1 -23020.874,E2 -23020.874} C_VEL
LIN {X 0,Y 171.577,Z 400.088,A -85,B 0,C 180,E1 -23025.772,E2 -23025.772} C_VEL
LIN {X 0,Y 171.885,Z 400.071,A -85,B 0,C 180,E1 -23030.586,E2 -23030.586} C_VEL
LIN {X 0,Y 171.816,Z 400.049,A -85,B 0,C 180,E1 -23035.307,E2 -23035.307} C_VEL
LIN {X 0,Y 172.331,Z 400.018,A -85,B 0,C 180,E1 -23039.999,E2 -23039.999} C_VEL
LIN {X 0,Y 171.819,Z 400.081,A -85,B 0,C 180,E1 -23044.692,E2 -23044.692} C_VEL
LIN {X 0,Y 171.885,Z 400.069,A -85,B 0,C 180,E1 -23049.413,E2 -23049.413} C_VEL
LIN {X 0,Y 171.608,Z 400.102,A -85,B 0,C 180,E1 -23054.224,E2 -23054.224} C_VEL
LIN {X 0,Y 171.572,Z 400.107,A -85,B 0,C 180,E1 -23059.59,E2 -23059.59} C_VEL
LIN {X 0,Y 171.466,Z 400.128,A -85,B 0,C 180,E1 -23065.616,E2 -23065.616} C_VEL
LIN {X 0,Y 171.436,Z 400.132,A -85,B 0,C 180,E1 -23070.586,E2 -23070.586} C_VEL
LIN {X 0,Y 171.4,Z 400.136,A -85,B 0,C 180,E1 -23075.033,E2 -23075.033} C_VEL
LIN {X 0,Y 171.424,Z 400.133,A -85,B 0,C 180,E1 -23078.837,E2 -23078.837} C_VEL
LIN {X 0,Y 171.411,Z 400.265,A -85,B 0,C 180,E1 -23083.7,E2 -23083.7} C_VEL
LIN {X 0,Y 172.546,Z 404.534,A -85,B 0,C 180,E1 -23086.445,E2 -23086.445} C_VEL
LIN {X 0,Y 174.963,Z 409.051,A -85,B 0,C 180,E1 -23087.321,E2 -23087.321} C_VEL
LIN {X 0,Y 181.483,Z 422.234,A -85,B 0,C 180,E1 -23089.569,E2 -23089.569} C_VEL
LIN {X 0,Y 187.884,Z 437.788,A -85,B 0,C 180,E1 -23091.688,E2 -23091.688} C_VEL
LIN {X 0,Y 189.801,Z 443.295,A -85,B 0,C 180,E1 -23092.323,E2 -23092.323} C_VEL
LIN {X 0,Y 192.115,Z 468.622,A -85,B 0,C 180,E1 -23093.88,E2 -23093.88} C_VEL
LIN {X 0,Y 189.878,Z 513.79,A -85,B 0,C 180,E1 -23095.485,E2 -23095.485} C_VEL
LIN {X 0,Y 188.538,Z 527.024,A -85,B 0,C 180,E1 -23096.326,E2 -23096.326} C_VEL
LIN {X 0,Y 186.601,Z 539.81,A -85,B 0,C 180,E1 -23097.541,E2 -23097.541} C_VEL
LIN {X 0,Y 185.293,Z 546.671,A -85,B 0,C 180,E1 -23098.394,E2 -23098.394} C_VEL
LIN {X 0,Y 183.608,Z 552.002,A -85,B 0,C 180,E1 -23099.079,E2 -23099.079} C_VEL
LIN {X 0,Y 179.151,Z 560.257,A -85,B 0,C 180,E1 -23100.121,E2 -23100.121} C_VEL
LIN {X 0,Y 174.467,Z 568.006,A -85,B 0,C 180,E1 -23101.386,E2 -23101.386} C_VEL
LIN {X 0,Y 172.453,Z 572.538,A -85,B 0,C 180,E1 -23102.406,E2 -23102.406} C_VEL
LIN {X 0,Y 169.985,Z 581.182,A -85,B 0,C 180,E1 -23104.927,E2 -23104.927} C_VEL
LIN {X 0,Y 168.023,Z 587.503,A -85,B 0,C 180,E1 -23107.156,E2 -23107.156} C_VEL
LIN {X 0,Y 166.456,Z 593.363,A -85,B 0,C 180,E1 -23109.616,E2 -23109.616} C_VEL
LIN {X 0,Y 164.457,Z 600.361,A -85,B 0,C 180,E1 -23113.235,E2 -23113.235} C_VEL
LIN {X 0,Y 162.859,Z 606.778,A -85,B 0,C 180,E1 -23117.54,E2 -23117.54} C_VEL
LIN {X 0,Y 162.19,Z 610.978,A -85,B 0,C 180,E1 -23121.277,E2 -23121.277} C_VEL
LIN {X 0,Y 161.986,Z 614.906,A -85,B 0,C 180,E1 -23126.27,E2 -23126.27} C_VEL
LIN {X 0,Y 162.183,Z 616.708,A -85,B 0,C 180,E1 -23130,E2 -23130} C_VEL
LIN {X 0,Y 161.942,Z 617.525,A -85,B 0,C 180,E1 -23133.482,E2 -23133.482} C_VEL
LIN {X 0,Y 162.003,Z 617.477,A -85,B 0,C 180,E1 -23137.478,E2 -23137.478} C_VEL
LIN {X 0,Y 162.357,Z 616.931,A -85,B 0,C 180,E1 -23139.971,E2 -23139.971} C_VEL
LIN {X 0,Y 163.822,Z 614.647,A -85,B 0,C 180,E1 -23144.916,E2 -23144.916} C_VEL
LIN {X 0,Y 165.77,Z 611.862,A -85,B 0,C 180,E1 -23148.54,E2 -23148.54} C_VEL
LIN {X 0,Y 168.362,Z 608.078,A -85,B 0,C 180,E1 -23152.066,E2 -23152.066} C_VEL
LIN {X 0,Y 171.591,Z 603.134,A -85,B 0,C 180,E1 -23155.516,E2 -23155.516} C_VEL
LIN {X 0,Y 175.219,Z 597.076,A -85,B 0,C 180,E1 -23158.771,E2 -23158.771} C_VEL
LIN {X 0,Y 179.656,Z 589.497,A -85,B 0,C 180,E1 -23161.877,E2 -23161.877} C_VEL
LIN {X 0,Y 183.832,Z 581.774,A -85,B 0,C 180,E1 -23164.325,E2 -23164.325} C_VEL
LIN {X 0,Y 188.777,Z 571.314,A -85,B 0,C 180,E1 -23166.892,E2 -23166.892} C_VEL
LIN {X 0,Y 193.151,Z 560.691,A -85,B 0,C 180,E1 -23168.877,E2 -23168.877} C_VEL
LIN {X 0,Y 196.72,Z 550.442,A -85,B 0,C 180,E1 -23170.355,E2 -23170.355} C_VEL
LIN {X 0,Y 200.233,Z 538.251,A -85,B 0,C 180,E1 -23171.657,E2 -23171.657} C_VEL
LIN {X 0,Y 203.102,Z 524.737,A -85,B 0,C 180,E1 -23172.684,E2 -23172.684} C_VEL
LIN {X 0,Y 204.889,Z 512.073,A -85,B 0,C 180,E1 -23173.315,E2 -23173.315} C_VEL
LIN {X 0,Y 207.224,Z 475.956,A -85,B 0,C 180,E1 -23174.494,E2 -23174.494} C_VEL
LIN {X 0,Y 206.787,Z 472.738,A -85,B 0,C 180,E1 -23174.796,E2 -23174.796} C_VEL
LIN {X 0,Y 201.941,Z 460.769,A -85,B 0,C 180,E1 -23177.032,E2 -23177.032} C_VEL
LIN {X 0,Y 196.519,Z 449.324,A -85,B 0,C 180,E1 -23179.695,E2 -23179.695} C_VEL
LIN {X 0,Y 191.378,Z 439.701,A -85,B 0,C 180,E1 -23182.462,E2 -23182.462} C_VEL
LIN {X 0,Y 186.644,Z 431.634,A -85,B 0,C 180,E1 -23185.294,E2 -23185.294} C_VEL
LIN {X 0,Y 183.1,Z 426.042,A -85,B 0,C 180,E1 -23187.659,E2 -23187.659} C_VEL
LIN {X 0,Y 179.279,Z 420.232,A -85,B 0,C 180,E1 -23190.528,E2 -23190.528} C_VEL
LIN {X 0,Y 176.073,Z 415.696,A -85,B 0,C 180,E1 -23193.268,E2 -23193.268} C_VEL
LIN {X 0,Y 175.353,Z 414.472,A -85,B 0,C 180,E1 -23193.964,E2 -23193.964} C_VEL
LIN {X 0,Y 172.283,Z 411.195,A -85,B 0,C 180,E1 -23197.041,E2 -23197.041} C_VEL
LIN {X 0,Y 170.475,Z 408.762,A -85,B 0,C 180,E1 -23199.251,E2 -23199.251} C_VEL
LIN {X 0,Y 169.847,Z 407.038,A -85,B 0,C 180,E1 -23200.235,E2 -23200.235} C_VEL
LIN {X 0,Y 166.578,Z 405.161,A -85,B 0,C 180,E1 -23205.337,E2 -23205.337} C_VEL
LIN {X 0,Y 165.135,Z 402.504,A -85,B 0,C 180,E1 -23209.392,E2 -23209.392} C_VEL
LIN {X 0,Y 164.822,Z 400.95,A -85,B 0,C 180,E1 -23211.263,E2 -23211.263} C_VEL
LIN {X 0,Y 165.047,Z 400.917,A -85,B 0,C 180,E1 -23217.56,E2 -23217.56} C_VEL
LIN {X 0,Y 165.293,Z 400.886,A -85,B 0,C 180,E1 -23220.001,E2 -23220.001} C_VEL
LIN {X 0,Y 165.119,Z 401.062,A -85,B 0,C 180,E1 -23221.677,E2 -23221.677} C_VEL
LIN {X 0,Y 165.634,Z 403.461,A -85,B 0,C 180,E1 -23223.954,E2 -23223.954} C_VEL
LIN {X 0,Y 168.106,Z 406.115,A -85,B 0,C 180,E1 -23229.021,E2 -23229.021} C_VEL
LIN {X 0,Y 170.079,Z 407.213,A -85,B 0,C 180,E1 -23231.757,E2 -23231.757} C_VEL
LIN {X 0,Y 171.411,Z 410.124,A -85,B 0,C 180,E1 -23233.637,E2 -23233.637} C_VEL
LIN {X 0,Y 174.057,Z 412.442,A -85,B 0,C 180,E1 -23236.419,E2 -23236.419} C_VEL
LIN {X 0,Y 174.86,Z 413.065,A -85,B 0,C 180,E1 -23237.168,E2 -23237.168} C_VEL
LIN {X 0,Y 176.76,Z 416.265,A -85,B 0,C 180,E1 -23238.999,E2 -23238.999} C_VEL
LIN {X 0,Y 179.225,Z 418.549,A -85,B 0,C 180,E1 -23240.967,E2 -23240.967} C_VEL
LIN {X 0,Y 181.569,Z 421.923,A -85,B 0,C 180,E1 -23242.773,E2 -23242.773} C_VEL
LIN {X 0,Y 183.3,Z 423.859,A -85,B 0,C 180,E1 -23243.966,E2 -23243.966} C_VEL
LIN {X 0,Y 186.977,Z 428.882,A -85,B 0,C 180,E1 -23246.36,E2 -23246.36} C_VEL
LIN {X 0,Y 190.502,Z 433.872,A -85,B 0,C 180,E1 -23248.434,E2 -23248.434} C_VEL
LIN {X 0,Y 193.572,Z 438.356,A -85,B 0,C 180,E1 -23250.099,E2 -23250.099} C_VEL
LIN {X 0,Y 199.261,Z 447.106,A -85,B 0,C 180,E1 -23252.915,E2 -23252.915} C_VEL
LIN {X 0,Y 204.631,Z 456.601,A -85,B 0,C 180,E1 -23255.346,E2 -23255.346} C_VEL
LIN {X 0,Y 208.12,Z 463.399,A -85,B 0,C 180,E1 -23256.828,E2 -23256.828} C_VEL
LIN {X 0,Y 205.517,Z 500.159,A -85,B 0,C 180,E1 -23257.992,E2 -23257.992} C_VEL
LIN {X 0,Y 203.736,Z 513.205,A -85,B 0,C 180,E1 -23258.727,E2 -23258.727} C_VEL
LIN {X 0,Y 201.272,Z 525.83,A -85,B 0,C 180,E1 -23259.81,E2 -23259.81} C_VEL
LIN {X 0,Y 198.108,Z 537.117,A -85,B 0,C 180,E1 -23261.076,E2 -23261.076} C_VEL
LIN {X 0,Y 194.617,Z 547.503,A -85,B 0,C 180,E1 -23262.628,E2 -23262.628} C_VEL
LIN {X 0,Y 190.679,Z 558.048,A -85,B 0,C 180,E1 -23264.74,E2 -23264.74} C_VEL
LIN {X 0,Y 186.198,Z 567.839,A -85,B 0,C 180,E1 -23267.204,E2 -23267.204} C_VEL
LIN {X 0,Y 182.114,Z 575.646,A -85,B 0,C 180,E1 -23269.73,E2 -23269.73} C_VEL
LIN {X 0,Y 178.185,Z 582.417,A -85,B 0,C 180,E1 -23272.504,E2 -23272.504} C_VEL
LIN {X 0,Y 174.38,Z 588.398,A -85,B 0,C 180,E1 -23275.652,E2 -23275.652} C_VEL
LIN {X 0,Y 170.919,Z 593.358,A -85,B 0,C 180,E1 -23279.071,E2 -23279.071} C_VEL
LIN {X 0,Y 168.015,Z 597.155,A -85,B 0,C 180,E1 -23282.605,E2 -23282.605} C_VEL
LIN {X 0,Y 166.387,Z 599.095,A -85,B 0,C 180,E1 -23285.015,E2 -23285.015} C_VEL
LIN {X 0,Y 165.078,Z 600.608,A -85,B 0,C 180,E1 -23287.471,E2 -23287.471} C_VEL
LIN {X 0,Y 163.681,Z 601.932,A -85,B 0,C 180,E1 -23290.845,E2 -23290.845} C_VEL
LIN {X 0,Y 162.514,Z 602.554,A -85,B 0,C 180,E1 -23294.962,E2 -23294.962} C_VEL
LIN {X 0,Y 162.069,Z 602.416,A -85,B 0,C 180,E1 -23297.478,E2 -23297.478} C_VEL
LIN {X 0,Y 161.956,Z 600.865,A -85,B 0,C 180,E1 -23302.52,E2 -23302.52} C_VEL
LIN {X 0,Y 162.226,Z 599.427,A -85,B 0,C 180,E1 -23305.157,E2 -23305.157} C_VEL
LIN {X 0,Y 162.659,Z 596.659,A -85,B 0,C 180,E1 -23308.762,E2 -23308.762} C_VEL
LIN {X 0,Y 163.543,Z 592.802,A -85,B 0,C 180,E1 -23312.463,E2 -23312.463} C_VEL
LIN {X 0,Y 164.906,Z 587.826,A -85,B 0,C 180,E1 -23316.116,E2 -23316.116} C_VEL
LIN {X 0,Y 166.791,Z 581.579,A -85,B 0,C 180,E1 -23319.703,E2 -23319.703} C_VEL
LIN {X 0,Y 169.238,Z 573.754,A -85,B 0,C 180,E1 -23323.203,E2 -23323.203} C_VEL
LIN {X 0,Y 172.183,Z 564.009,A -85,B 0,C 180,E1 -23326.601,E2 -23326.601} C_VEL
LIN {X 0,Y 175.11,Z 553.85,A -85,B 0,C 180,E1 -23329.336,E2 -23329.336} C_VEL
LIN {X 0,Y 177.953,Z 542.376,A -85,B 0,C 180,E1 -23331.731,E2 -23331.731} C_VEL
LIN {X 0,Y 180.217,Z 531.118,A -85,B 0,C 180,E1 -23333.56,E2 -23333.56} C_VEL
LIN {X 0,Y 182.146,Z 519.582,A -85,B 0,C 180,E1 -23334.961,E2 -23334.961} C_VEL
LIN {X 0,Y 183.72,Z 506.261,A -85,B 0,C 180,E1 -23336.105,E2 -23336.105} C_VEL
LIN {X 0,Y 184.604,Z 494.191,A -85,B 0,C 180,E1 -23336.762,E2 -23336.762} C_VEL
LIN {X 0,Y 187.099,Z 442.945,A -85,B 0,C 180,E1 -23338.598,E2 -23338.598} C_VEL
LIN {X 0,Y 179.921,Z 427.655,A -85,B 0,C 180,E1 -23340.89,E2 -23340.89} C_VEL
LIN {X 0,Y 173.019,Z 415.489,A -85,B 0,C 180,E1 -23343.213,E2 -23343.213} C_VEL
LIN {X 0,Y 166.567,Z 405.372,A -85,B 0,C 180,E1 -23345.561,E2 -23345.561} C_VEL
LIN {X 0,Y 164.82,Z 402.914,A -85,B 0,C 180,E1 -23346.228,E2 -23346.228} C_VEL
LIN {X 0,Y 164.309,Z 401.016,A -85,B 0,C 180,E1 -23346.558,E2 -23346.558} C_VEL
LIN {X 0,Y 164.295,Z 401.007,A -85,B 0,C 180,E1 -23349.914,E2 -23349.914} C_VEL
LIN {X 0,Y 164.307,Z 401.015,A -85,B 0,C 180,E1 -23353.351,E2 -23353.351} C_VEL
LIN {X 0,Y 164.357,Z 400.991,A -85,B 0,C 180,E1 -23356.829,E2 -23356.829} C_VEL
LIN {X 0,Y 164.374,Z 401.006,A -85,B 0,C 180,E1 -23360.317,E2 -23360.317} C_VEL
LIN {X 0,Y 164.346,Z 400.989,A -85,B 0,C 180,E1 -23364.339,E2 -23364.339} C_VEL
LIN {X 0,Y 164.388,Z 401.008,A -85,B 0,C 180,E1 -23369.133,E2 -23369.133} C_VEL
LIN {X 0,Y 164.416,Z 400.977,A -85,B 0,C 180,E1 -23374.693,E2 -23374.693} C_VEL
LIN {X 0,Y 164.519,Z 400.991,A -85,B 0,C 180,E1 -23380.016,E2 -23380.016} C_VEL
LIN {X 0,Y 164.527,Z 400.961,A -85,B 0,C 180,E1 -23385.149,E2 -23385.149} C_VEL
LIN {X 0,Y 164.799,Z 400.956,A -85,B 0,C 180,E1 -23390.178,E2 -23390.178} C_VEL
LIN {X 0,Y 164.847,Z 400.934,A -85,B 0,C 180,E1 -23392.651,E2 -23392.651} C_VEL
LIN {X 0,Y 165.045,Z 400.911,A -85,B 0,C 180,E1 -23397.559,E2 -23397.559} C_VEL
LIN {X 0,Y 165.293,Z 400.894,A -85,B 0,C 180,E1 -23399.999,E2 -23399.999} C_VEL
LIN {X 0,Y 164.769,Z 400.959,A -85,B 0,C 180,E1 -23404.893,E2 -23404.893} C_VEL
LIN {X 0,Y 164.848,Z 400.947,A -85,B 0,C 180,E1 -23407.348,E2 -23407.348} C_VEL
LIN {X 0,Y 164.751,Z 400.963,A -85,B 0,C 180,E1 -23411.151,E2 -23411.151} C_VEL
LIN {X 0,Y 164.523,Z 400.991,A -85,B 0,C 180,E1 -23417.398,E2 -23417.398} C_VEL
LIN {X 0,Y 164.517,Z 400.988,A -85,B 0,C 180,E1 -23419.983,E2 -23419.983} C_VEL
LIN {X 0,Y 164.39,Z 401.01,A -85,B 0,C 180,E1 -23426.134,E2 -23426.134} C_VEL
LIN {X 0,Y 164.371,Z 401.012,A -85,B 0,C 180,E1 -23431.227,E2 -23431.227} C_VEL
LIN {X 0,Y 164.345,Z 401.014,A -85,B 0,C 180,E1 -23436.776,E2 -23436.776} C_VEL
LIN {X 0,Y 164.402,Z 401.035,A -85,B 0,C 180,E1 -23442.218,E2 -23442.218} C_VEL
LIN {X 0,Y 165.13,Z 404.01,A -85,B 0,C 180,E1 -23444.288,E2 -23444.288} C_VEL
LIN {X 0,Y 167.719,Z 408.728,A -85,B 0,C 180,E1 -23445.32,E2 -23445.32} C_VEL
LIN {X 0,Y 174.521,Z 421.938,A -85,B 0,C 180,E1 -23447.869,E2 -23447.869} C_VEL
LIN {X 0,Y 180.749,Z 436.479,A -85,B 0,C 180,E1 -23450.087,E2 -23450.087} C_VEL
LIN {X 0,Y 184.018,Z 445.509,A -85,B 0,C 180,E1 -23451.233,E2 -23451.233} C_VEL
LIN {X 0,Y 186.082,Z 469.674,A -85,B 0,C 180,E1 -23452.767,E2 -23452.767} C_VEL
LIN {X 0,Y 183.771,Z 513.763,A -85,B 0,C 180,E1 -23454.375,E2 -23454.375} C_VEL
LIN {X 0,Y 182.336,Z 527.287,A -85,B 0,C 180,E1 -23455.269,E2 -23455.269} C_VEL
LIN {X 0,Y 180.421,Z 539.35,A -85,B 0,C 180,E1 -23456.452,E2 -23456.452} C_VEL
LIN {X 0,Y 177.943,Z 551.528,A -85,B 0,C 180,E1 -23458.113,E2 -23458.113} C_VEL
LIN {X 0,Y 175.058,Z 563.106,A -85,B 0,C 180,E1 -23460.211,E2 -23460.211} C_VEL
LIN {X 0,Y 172.453,Z 572.538,A -85,B 0,C 180,E1 -23462.406,E2 -23462.406} C_VEL
LIN {X 0,Y 170.477,Z 576.981,A -85,B 0,C 180,E1 -23463.527,E2 -23463.527} C_VEL
LIN {X 0,Y 165.848,Z 583.779,A -85,B 0,C 180,E1 -23465.402,E2 -23465.402} C_VEL
LIN {X 0,Y 161.3,Z 589.992,A -85,B 0,C 180,E1 -23467.575,E2 -23467.575} C_VEL
LIN {X 0,Y 159.492,Z 593.517,A -85,B 0,C 180,E1 -23469.138,E2 -23469.138} C_VEL
LIN {X 0,Y 157.307,Z 600.764,A -85,B 0,C 180,E1 -23473.118,E2 -23473.118} C_VEL
LIN {X 0,Y 155.892,Z 606.217,A -85,B 0,C 180,E1 -23476.973,E2 -23476.973} C_VEL
LIN {X 0,Y 155.16,Z 610.471,A -85,B 0,C 180,E1 -23480.878,E2 -23480.878} C_VEL
LIN {X 0,Y 154.922,Z 614.637,A -85,B 0,C 180,E1 -23486.393,E2 -23486.393} C_VEL
LIN {X 0,Y 155.102,Z 616.32,A -85,B 0,C 180,E1 -23490,E2 -23490} C_VEL
LIN {X 0,Y 154.875,Z 617.106,A -85,B 0,C 180,E1 -23493.319,E2 -23493.319} C_VEL
LIN {X 0,Y 154.948,Z 617.153,A -85,B 0,C 180,E1 -23497.82,E2 -23497.82} C_VEL
LIN {X 0,Y 155.332,Z 616.65,A -85,B 0,C 180,E1 -23500.427,E2 -23500.427} C_VEL
LIN {X 0,Y 156.931,Z 614.411,A -85,B 0,C 180,E1 -23505.587,E2 -23505.587} C_VEL
LIN {X 0,Y 159.029,Z 611.674,A -85,B 0,C 180,E1 -23509.356,E2 -23509.356} C_VEL
LIN {X 0,Y 161.79,Z 607.941,A -85,B 0,C 180,E1 -23513.013,E2 -23513.013} C_VEL
LIN {X 0,Y 165.523,Z 602.519,A -85,B 0,C 180,E1 -23516.92,E2 -23516.92} C_VEL
LIN {X 0,Y 169.739,Z 595.933,A -85,B 0,C 180,E1 -23520.477,E2 -23520.477} C_VEL
LIN {X 0,Y 174.502,Z 588.127,A -85,B 0,C 180,E1 -23523.626,E2 -23523.626} C_VEL
LIN {X 0,Y 179.823,Z 578.404,A -85,B 0,C 180,E1 -23526.584,E2 -23526.584} C_VEL
LIN {X 0,Y 184.142,Z 569.45,A -85,B 0,C 180,E1 -23528.679,E2 -23528.679} C_VEL
LIN {X 0,Y 188.208,Z 559.8,A -85,B 0,C 180,E1 -23530.451,E2 -23530.451} C_VEL
LIN {X 0,Y 191.949,Z 549.413,A -85,B 0,C 180,E1 -23531.927,E2 -23531.927} C_VEL
LIN {X 0,Y 195.302,Z 538.069,A -85,B 0,C 180,E1 -23533.134,E2 -23533.134} C_VEL
LIN {X 0,Y 198.292,Z 524.477,A -85,B 0,C 180,E1 -23534.172,E2 -23534.172} C_VEL
LIN {X 0,Y 200.153,Z 511.705,A -85,B 0,C 180,E1 -23534.811,E2 -23534.811} C_VEL
LIN {X 0,Y 202.495,Z 477.031,A -85,B 0,C 180,E1 -23535.955,E2 -23535.955} C_VEL
LIN {X 0,Y 201.417,Z 473.516,A -85,B 0,C 180,E1 -23536.51,E2 -23536.51} C_VEL
LIN {X 0,Y 196.452,Z 461.579,A -85,B 0,C 180,E1 -23538.986,E2 -23538.986} C_VEL
LIN {X 0,Y 191.53,Z 451.196,A -85,B 0,C 180,E1 -23541.64,E2 -23541.64} C_VEL
LIN {X 0,Y 186.879,Z 442.43,A -85,B 0,C 180,E1 -23544.39,E2 -23544.39} C_VEL
LIN {X 0,Y 183.492,Z 436.699,A -85,B 0,C 180,E1 -23546.59,E2 -23546.59} C_VEL
LIN {X 0,Y 180.806,Z 432.226,A -85,B 0,C 180,E1 -23548.506,E2 -23548.506} C_VEL
LIN {X 0,Y 177.163,Z 426.497,A -85,B 0,C 180,E1 -23551.396,E2 -23551.396} C_VEL
LIN {X 0,Y 173.97,Z 421.679,A -85,B 0,C 180,E1 -23554.313,E2 -23554.313} C_VEL
LIN {X 0,Y 172.353,Z 419.69,A -85,B 0,C 180,E1 -23555.936,E2 -23555.936} C_VEL
LIN {X 0,Y 169.026,Z 415.463,A -85,B 0,C 180,E1 -23559.919,E2 -23559.919} C_VEL
LIN {X 0,Y 168.343,Z 413.854,A -85,B 0,C 180,E1 -23561.009,E2 -23561.009} C_VEL
LIN {X 0,Y 165.303,Z 411.85,A -85,B 0,C 180,E1 -23566.164,E2 -23566.164} C_VEL
LIN {X 0,Y 164.018,Z 408.954,A -85,B 0,C 180,E1 -23570.443,E2 -23570.443} C_VEL
LIN {X 0,Y 163.893,Z 408.089,A -85,B 0,C 180,E1 -23571.369,E2 -23571.369} C_VEL
LIN {X 0,Y 164.092,Z 407.978,A -85,B 0,C 180,E1 -23581.074,E2 -23581.074} C_VEL
LIN {X 0,Y 164.643,Z 410.498,A -85,B 0,C 180,E1 -23583.672,E2 -23583.672} C_VEL
LIN {X 0,Y 167.427,Z 413.303,A -85,B 0,C 180,E1 -23589.362,E2 -23589.362} C_VEL
LIN {X 0,Y 168.63,Z 414.129,A -85,B 0,C 180,E1 -23591.087,E2 -23591.087} C_VEL
LIN {X 0,Y 170.106,Z 417.032,A -85,B 0,C 180,E1 -23593.211,E2 -23593.211} C_VEL
LIN {X 0,Y 172.774,Z 419.352,A -85,B 0,C 180,E1 -23596.089,E2 -23596.089} C_VEL
LIN {X 0,Y 173.433,Z 420.406,A -85,B 0,C 180,E1 -23596.782,E2 -23596.782} C_VEL
LIN {X 0,Y 175.731,Z 423.595,A -85,B 0,C 180,E1 -23598.963,E2 -23598.963} C_VEL
LIN {X 0,Y 177.26,Z 425.08,A -85,B 0,C 180,E1 -23600.224,E2 -23600.224} C_VEL
LIN {X 0,Y 179.893,Z 428.73,A -85,B 0,C 180,E1 -23602.315,E2 -23602.315} C_VEL
LIN {X 0,Y 181.125,Z 430.279,A -85,B 0,C 180,E1 -23603.21,E2 -23603.21} C_VEL
LIN {X 0,Y 184.47,Z 434.918,A -85,B 0,C 180,E1 -23605.493,E2 -23605.493} C_VEL
LIN {X 0,Y 189.505,Z 442.211,A -85,B 0,C 180,E1 -23608.541,E2 -23608.541} C_VEL
LIN {X 0,Y 195.732,Z 452.073,A -85,B 0,C 180,E1 -23611.848,E2 -23611.848} C_VEL
LIN {X 0,Y 201.343,Z 462.317,A -85,B 0,C 180,E1 -23614.534,E2 -23614.534} C_VEL
LIN {X 0,Y 203.247,Z 465.98,A -85,B 0,C 180,E1 -23615.387,E2 -23615.387} C_VEL
LIN {X 0,Y 200.729,Z 500.804,A -85,B 0,C 180,E1 -23616.528,E2 -23616.528} C_VEL
LIN {X 0,Y 198.86,Z 513.776,A -85,B 0,C 180,E1 -23617.264,E2 -23617.264} C_VEL
LIN {X 0,Y 196.462,Z 525.727,A -85,B 0,C 180,E1 -23618.303,E2 -23618.303} C_VEL
LIN {X 0,Y 192.906,Z 537.942,A -85,B 0,C 180,E1 -23619.681,E2 -23619.681} C_VEL
LIN {X 0,Y 189.283,Z 548.237,A -85,B 0,C 180,E1 -23621.249,E2 -23621.249} C_VEL
LIN {X 0,Y 185.232,Z 558.588,A -85,B 0,C 180,E1 -23623.365,E2 -23623.365} C_VEL
LIN {X 0,Y 180.941,Z 567.559,A -85,B 0,C 180,E1 -23625.643,E2 -23625.643} C_VEL
LIN {X 0,Y 176.626,Z 575.493,A -85,B 0,C 180,E1 -23628.205,E2 -23628.205} C_VEL
LIN {X 0,Y 172.292,Z 582.641,A -85,B 0,C 180,E1 -23631.172,E2 -23631.172} C_VEL
LIN {X 0,Y 168.435,Z 588.415,A -85,B 0,C 180,E1 -23634.258,E2 -23634.258} C_VEL
LIN {X 0,Y 164.734,Z 593.443,A -85,B 0,C 180,E1 -23637.773,E2 -23637.773} C_VEL
LIN {X 0,Y 161.598,Z 597.304,A -85,B 0,C 180,E1 -23641.42,E2 -23641.42} C_VEL
LIN {X 0,Y 159.832,Z 599.275,A -85,B 0,C 180,E1 -23643.915,E2 -23643.915} C_VEL
LIN {X 0,Y 158.385,Z 600.821,A -85,B 0,C 180,E1 -23646.463,E2 -23646.463} C_VEL
LIN {X 0,Y 156.714,Z 602.312,A -85,B 0,C 180,E1 -23650.353,E2 -23650.353} C_VEL
LIN {X 0,Y 155.561,Z 602.878,A -85,B 0,C 180,E1 -23654.272,E2 -23654.272} C_VEL
LIN {X 0,Y 155.043,Z 602.777,A -85,B 0,C 180,E1 -23656.901,E2 -23656.901} C_VEL
LIN {X 0,Y 154.823,Z 602.245,A -85,B 0,C 180,E1 -23659.539,E2 -23659.539} C_VEL
LIN {X 0,Y 155.101,Z 599.966,A -85,B 0,C 180,E1 -23664.801,E2 -23664.801} C_VEL
LIN {X 0,Y 155.566,Z 597.18,A -85,B 0,C 180,E1 -23668.706,E2 -23668.706} C_VEL
LIN {X 0,Y 156.436,Z 593.388,A -85,B 0,C 180,E1 -23672.575,E2 -23672.575} C_VEL
LIN {X 0,Y 157.856,Z 588.478,A -85,B 0,C 180,E1 -23676.39,E2 -23676.39} C_VEL
LIN {X 0,Y 159.822,Z 582.306,A -85,B 0,C 180,E1 -23680.131,E2 -23680.131} C_VEL
LIN {X 0,Y 162.366,Z 574.608,A -85,B 0,C 180,E1 -23683.772,E2 -23683.772} C_VEL
LIN {X 0,Y 165.418,Z 564.968,A -85,B 0,C 180,E1 -23687.301,E2 -23687.301} C_VEL
LIN {X 0,Y 168.455,Z 554.995,A -85,B 0,C 180,E1 -23690.132,E2 -23690.132} C_VEL
LIN {X 0,Y 171.4,Z 543.714,A -85,B 0,C 180,E1 -23692.606,E2 -23692.606} C_VEL
LIN {X 0,Y 173.79,Z 532.686,A -85,B 0,C 180,E1 -23694.488,E2 -23694.488} C_VEL
LIN {X 0,Y 175.968,Z 520.428,A -85,B 0,C 180,E1 -23696.06,E2 -23696.06} C_VEL
LIN {X 0,Y 177.592,Z 507.439,A -85,B 0,C 180,E1 -23697.229,E2 -23697.229} C_VEL
LIN {X 0,Y 178.566,Z 495.047,A -85,B 0,C 180,E1 -23697.942,E2 -23697.942} C_VEL
LIN {X 0,Y 181.124,Z 444.936,A -85,B 0,C 180,E1 -23699.784,E2 -23699.784} C_VEL
LIN {X 0,Y 173.805,Z 429.458,A -85,B 0,C 180,E1 -23702.287,E2 -23702.287} C_VEL
LIN {X 0,Y 166.971,Z 417.583,A -85,B 0,C 180,E1 -23704.764,E2 -23704.764} C_VEL
LIN {X 0,Y 162.352,Z 410.422,A -85,B 0,C 180,E1 -23706.562,E2 -23706.562} C_VEL
LIN {X 0,Y 160.166,Z 406.935,A -85,B 0,C 180,E1 -23707.474,E2 -23707.474} C_VEL
LIN {X 0,Y 157.975,Z 404.294,A -85,B 0,C 180,E1 -23708.374,E2 -23708.374} C_VEL
LIN {X 0,Y 157.213,Z 401.899,A -85,B 0,C 180,E1 -23708.854,E2 -23708.854} C_VEL
LIN {X 0,Y 157.217,Z 401.899,A -85,B 0,C 180,E1 -23714.336,E2 -23714.336} C_VEL
LIN {X 0,Y 157.279,Z 401.882,A -85,B 0,C 180,E1 -23719.431,E2 -23719.431} C_VEL
LIN {X 0,Y 157.293,Z 401.866,A -85,B 0,C 180,E1 -23724.488,E2 -23724.488} C_VEL
LIN {X 0,Y 157.292,Z 401.886,A -85,B 0,C 180,E1 -23728.095,E2 -23728.095} C_VEL
LIN {X 0,Y 157.319,Z 401.862,A -85,B 0,C 180,E1 -23733.465,E2 -23733.465} C_VEL
LIN {X 0,Y 157.445,Z 401.873,A -85,B 0,C 180,E1 -23739.615,E2 -23739.615} C_VEL
LIN {X 0,Y 157.46,Z 401.838,A -85,B 0,C 180,E1 -23744.466,E2 -23744.466} C_VEL
LIN {X 0,Y 157.723,Z 401.837,A -85,B 0,C 180,E1 -23749.732,E2 -23749.732} C_VEL
LIN {X 0,Y 157.804,Z 401.814,A -85,B 0,C 180,E1 -23752.321,E2 -23752.321} C_VEL
LIN {X 0,Y 158.255,Z 401.771,A -85,B 0,C 180,E1 -23759.999,E2 -23759.999} C_VEL
LIN {X 0,Y 157.805,Z 401.822,A -85,B 0,C 180,E1 -23767.678,E2 -23767.678} C_VEL
LIN {X 0,Y 157.68,Z 401.844,A -85,B 0,C 180,E1 -23771.321,E2 -23771.321} C_VEL
LIN {X 0,Y 157.484,Z 401.866,A -85,B 0,C 180,E1 -23775.531,E2 -23775.531} C_VEL
LIN {X 0,Y 157.413,Z 401.878,A -85,B 0,C 180,E1 -23780.926,E2 -23780.926} C_VEL
LIN {X 0,Y 157.311,Z 401.89,A -85,B 0,C 180,E1 -23786.684,E2 -23786.684} C_VEL
LIN {X 0,Y 157.274,Z 401.897,A -85,B 0,C 180,E1 -23792.427,E2 -23792.427} C_VEL
LIN {X 0,Y 157.319,Z 401.89,A -85,B 0,C 180,E1 -23796.476,E2 -23796.476} C_VEL
LIN {X 0,Y 157.324,Z 401.981,A -85,B 0,C 180,E1 -23800.686,E2 -23800.686} C_VEL
LIN {X 0,Y 157.839,Z 403.726,A -85,B 0,C 180,E1 -23801.904,E2 -23801.904} C_VEL
LIN {X 0,Y 160.184,Z 408.015,A -85,B 0,C 180,E1 -23802.957,E2 -23802.957} C_VEL
LIN {X 0,Y 164.472,Z 415.837,A -85,B 0,C 180,E1 -23804.76,E2 -23804.76} C_VEL
LIN {X 0,Y 169.95,Z 426.704,A -85,B 0,C 180,E1 -23806.918,E2 -23806.918} C_VEL
LIN {X 0,Y 175.842,Z 440.866,A -85,B 0,C 180,E1 -23809.153,E2 -23809.153} C_VEL
LIN {X 0,Y 178.292,Z 447.783,A -85,B 0,C 180,E1 -23810.072,E2 -23810.072} C_VEL
LIN {X 0,Y 180.13,Z 469.889,A -85,B 0,C 180,E1 -23811.542,E2 -23811.542} C_VEL
LIN {X 0,Y 177.776,Z 513.469,A -85,B 0,C 180,E1 -23813.178,E2 -23813.178} C_VEL
LIN {X 0,Y 176.262,Z 526.767,A -85,B 0,C 180,E1 -23814.066,E2 -23814.066} C_VEL
LIN {X 0,Y 174.322,Z 538.892,A -85,B 0,C 180,E1 -23815.288,E2 -23815.288} C_VEL
LIN {X 0,Y 171.879,Z 550.296,A -85,B 0,C 180,E1 -23816.847,E2 -23816.847} C_VEL
LIN {X 0,Y 169.258,Z 560.745,A -85,B 0,C 180,E1 -23818.734,E2 -23818.734} C_VEL
LIN {X 0,Y 166.141,Z 571.524,A -85,B 0,C 180,E1 -23821.238,E2 -23821.238} C_VEL
LIN {X 0,Y 163.534,Z 580.348,A -85,B 0,C 180,E1 -23823.865,E2 -23823.865} C_VEL
LIN {X 0,Y 161.008,Z 588.458,A -85,B 0,C 180,E1 -23826.869,E2 -23826.869} C_VEL
LIN {X 0,Y 159.492,Z 593.517,A -85,B 0,C 180,E1 -23829.138,E2 -23829.138} C_VEL
LIN {X 0,Y 157.715,Z 596.863,A -85,B 0,C 180,E1 -23830.792,E2 -23830.792} C_VEL
LIN {X 0,Y 153.418,Z 601.758,A -85,B 0,C 180,E1 -23833.559,E2 -23833.559} C_VEL
LIN {X 0,Y 149.513,Z 605.962,A -85,B 0,C 180,E1 -23836.613,E2 -23836.613} C_VEL
LIN {X 0,Y 148.389,Z 608.233,A -85,B 0,C 180,E1 -23838.657,E2 -23838.657} C_VEL
LIN {X 0,Y 147.817,Z 612.235,A -85,B 0,C 180,E1 -23843.174,E2 -23843.174} C_VEL
LIN {X 0,Y 147.863,Z 614.767,A -85,B 0,C 180,E1 -23847.276,E2 -23847.276} C_VEL
LIN {X 0,Y 148.022,Z 615.93,A -85,B 0,C 180,E1 -23850,E2 -23850} C_VEL
LIN {X 0,Y 147.795,Z 616.667,A -85,B 0,C 180,E1 -23853.036,E2 -23853.036} C_VEL
LIN {X 0,Y 147.891,Z 616.829,A -85,B 0,C 180,E1 -23858.196,E2 -23858.196} C_VEL
LIN {X 0,Y 148.326,Z 616.361,A -85,B 0,C 180,E1 -23860.925,E2 -23860.925} C_VEL
LIN {X 0,Y 150.067,Z 614.177,A -85,B 0,C 180,E1 -23866.319,E2 -23866.319} C_VEL
LIN {X 0,Y 152.327,Z 611.489,A -85,B 0,C 180,E1 -23870.244,E2 -23870.244} C_VEL
LIN {X 0,Y 155.269,Z 607.807,A -85,B 0,C 180,E1 -23874.039,E2 -23874.039} C_VEL
LIN {X 0,Y 158.922,Z 602.846,A -85,B 0,C 180,E1 -23877.816,E2 -23877.816} C_VEL
LIN {X 0,Y 163.657,Z 595.915,A -85,B 0,C 180,E1 -23881.739,E2 -23881.739} C_VEL
LIN {X 0,Y 168.627,Z 588.213,A -85,B 0,C 180,E1 -23884.964,E2 -23884.964} C_VEL
LIN {X 0,Y 174.193,Z 578.574,A -85,B 0,C 180,E1 -23887.971,E2 -23887.971} C_VEL
LIN {X 0,Y 178.672,Z 569.721,A -85,B 0,C 180,E1 -23890.097,E2 -23890.097} C_VEL
LIN {X 0,Y 182.886,Z 560.196,A -85,B 0,C 180,E1 -23891.888,E2 -23891.888} C_VEL
LIN {X 0,Y 187.339,Z 548.332,A -85,B 0,C 180,E1 -23893.576,E2 -23893.576} C_VEL
LIN {X 0,Y 190.712,Z 537.061,A -85,B 0,C 180,E1 -23894.761,E2 -23894.761} C_VEL
LIN {X 0,Y 193.738,Z 523.495,A -85,B 0,C 180,E1 -23895.786,E2 -23895.786} C_VEL
LIN {X 0,Y 195.584,Z 510.998,A -85,B 0,C 180,E1 -23896.394,E2 -23896.394} C_VEL
LIN {X 0,Y 197.843,Z 478.931,A -85,B 0,C 180,E1 -23897.46,E2 -23897.46} C_VEL
LIN {X 0,Y 193.356,Z 467.465,A -85,B 0,C 180,E1 -23899.847,E2 -23899.847} C_VEL
LIN {X 0,Y 188.426,Z 456.639,A -85,B 0,C 180,E1 -23902.663,E2 -23902.663} C_VEL
LIN {X 0,Y 183.708,Z 447.469,A -85,B 0,C 180,E1 -23905.643,E2 -23905.643} C_VEL
LIN {X 0,Y 180.687,Z 442.13,A -85,B 0,C 180,E1 -23907.751,E2 -23907.751} C_VEL
LIN {X 0,Y 178.266,Z 437.978,A -85,B 0,C 180,E1 -23909.597,E2 -23909.597} C_VEL
LIN {X 0,Y 174.998,Z 432.617,A -85,B 0,C 180,E1 -23912.365,E2 -23912.365} C_VEL
LIN {X 0,Y 171.957,Z 427.727,A -85,B 0,C 180,E1 -23915.349,E2 -23915.349} C_VEL
LIN {X 0,Y 169.236,Z 424.5,A -85,B 0,C 180,E1 -23918.374,E2 -23918.374} C_VEL
LIN {X 0,Y 167.358,Z 421.629,A -85,B 0,C 180,E1 -23920.991,E2 -23920.991} C_VEL
LIN {X 0,Y 167.06,Z 420.851,A -85,B 0,C 180,E1 -23921.511,E2 -23921.511} C_VEL
LIN {X 0,Y 164.013,Z 418.455,A -85,B 0,C 180,E1 -23927.157,E2 -23927.157} C_VEL
LIN {X 0,Y 162.924,Z 415.081,A -85,B 0,C 180,E1 -23931.858,E2 -23931.858} C_VEL
LIN {X 0,Y 163.105,Z 415.021,A -85,B 0,C 180,E1 -23940.618,E2 -23940.618} C_VEL
LIN {X 0,Y 163.706,Z 417.613,A -85,B 0,C 180,E1 -23943.539,E2 -23943.539} C_VEL
LIN {X 0,Y 166.757,Z 420.518,A -85,B 0,C 180,E1 -23949.706,E2 -23949.706} C_VEL
LIN {X 0,Y 167.248,Z 420.965,A -85,B 0,C 180,E1 -23950.443,E2 -23950.443} C_VEL
LIN {X 0,Y 169.04,Z 424.216,A -85,B 0,C 180,E1 -23953.066,E2 -23953.066} C_VEL
LIN {X 0,Y 171.422,Z 426.391,A -85,B 0,C 180,E1 -23955.704,E2 -23955.704} C_VEL
LIN {X 0,Y 173.637,Z 429.767,A -85,B 0,C 180,E1 -23957.977,E2 -23957.977} C_VEL
LIN {X 0,Y 175.516,Z 431.879,A -85,B 0,C 180,E1 -23959.633,E2 -23959.633} C_VEL
LIN {X 0,Y 179.114,Z 436.853,A -85,B 0,C 180,E1 -23962.532,E2 -23962.532} C_VEL
LIN {X 0,Y 182.168,Z 441.189,A -85,B 0,C 180,E1 -23964.712,E2 -23964.712} C_VEL
LIN {X 0,Y 186.808,Z 448.144,A -85,B 0,C 180,E1 -23967.672,E2 -23967.672} C_VEL
LIN {X 0,Y 192.54,Z 457.532,A -85,B 0,C 180,E1 -23970.885,E2 -23970.885} C_VEL
LIN {X 0,Y 197.622,Z 467.085,A -85,B 0,C 180,E1 -23973.466,E2 -23973.466} C_VEL
LIN {X 0,Y 198.559,Z 468.882,A -85,B 0,C 180,E1 -23973.913,E2 -23973.913} C_VEL
LIN {X 0,Y 196.103,Z 501.12,A -85,B 0,C 180,E1 -23974.974,E2 -23974.974} C_VEL
LIN {X 0,Y 194.167,Z 514.125,A -85,B 0,C 180,E1 -23975.716,E2 -23975.716} C_VEL
LIN {X 0,Y 191.513,Z 526.744,A -85,B 0,C 180,E1 -23976.828,E2 -23976.828} C_VEL
LIN {X 0,Y 187.82,Z 538.766,A -85,B 0,C 180,E1 -23978.208,E2 -23978.208} C_VEL
LIN {X 0,Y 183.576,Z 550.286,A -85,B 0,C 180,E1 -23980.034,E2 -23980.034} C_VEL
LIN {X 0,Y 179.205,Z 560.618,A -85,B 0,C 180,E1 -23982.25,E2 -23982.25} C_VEL
LIN {X 0,Y 173.956,Z 570.663,A -85,B 0,C 180,E1 -23985.009,E2 -23985.009} C_VEL
LIN {X 0,Y 168.731,Z 579.455,A -85,B 0,C 180,E1 -23988.209,E2 -23988.209} C_VEL
LIN {X 0,Y 164.061,Z 586.414,A -85,B 0,C 180,E1 -23991.601,E2 -23991.601} C_VEL
LIN {X 0,Y 159.894,Z 591.948,A -85,B 0,C 180,E1 -23995.153,E2 -23995.153} C_VEL
LIN {X 0,Y 156.687,Z 595.846,A -85,B 0,C 180,E1 -23998.456,E2 -23998.456} C_VEL
LIN {X 0,Y 153.341,Z 599.457,A -85,B 0,C 180,E1 -24002.722,E2 -24002.722} C_VEL
LIN {X 0,Y 151.768,Z 601.033,A -85,B 0,C 180,E1 -24005.37,E2 -24005.37} C_VEL
LIN {X 0,Y 149.754,Z 602.695,A -85,B 0,C 180,E1 -24009.822,E2 -24009.822} C_VEL
LIN {X 0,Y 148.641,Z 603.202,A -85,B 0,C 180,E1 -24013.52,E2 -24013.52} C_VEL
LIN {X 0,Y 148.033,Z 603.13,A -85,B 0,C 180,E1 -24016.268,E2 -24016.268} C_VEL
LIN {X 0,Y 147.76,Z 602.652,A -85,B 0,C 180,E1 -24019.033,E2 -24019.033} C_VEL
LIN {X 0,Y 147.735,Z 601.739,A -85,B 0,C 180,E1 -24021.795,E2 -24021.795} C_VEL
LIN {X 0,Y 148.079,Z 599.998,A -85,B 0,C 180,E1 -24025.347,E2 -24025.347} C_VEL
LIN {X 0,Y 148.674,Z 596.59,A -85,B 0,C 180,E1 -24030,E2 -24030} C_VEL
LIN {X 0,Y 149.825,Z 592.497,A -85,B 0,C 180,E1 -24034.035,E2 -24034.035} C_VEL
LIN {X 0,Y 151.794,Z 586.243,A -85,B 0,C 180,E1 -24038.654,E2 -24038.654} C_VEL
LIN {X 0,Y 154.107,Z 579.442,A -85,B 0,C 180,E1 -24042.51,E2 -24042.51} C_VEL
LIN {X 0,Y 157.009,Z 570.953,A -85,B 0,C 180,E1 -24046.246,E2 -24046.246} C_VEL
LIN {X 0,Y 159.914,Z 562.223,A -85,B 0,C 180,E1 -24049.245,E2 -24049.245} C_VEL
LIN {X 0,Y 163.235,Z 551.472,A -85,B 0,C 180,E1 -24052.131,E2 -24052.131} C_VEL
LIN {X 0,Y 165.995,Z 540.727,A -85,B 0,C 180,E1 -24054.38,E2 -24054.38} C_VEL
LIN {X 0,Y 168.542,Z 528.693,A -85,B 0,C 180,E1 -24056.298,E2 -24056.298} C_VEL
LIN {X 0,Y 170.639,Z 516.124,A -85,B 0,C 180,E1 -24057.769,E2 -24057.769} C_VEL
LIN {X 0,Y 172.063,Z 503.817,A -85,B 0,C 180,E1 -24058.764,E2 -24058.764} C_VEL
LIN {X 0,Y 173.049,Z 489.244,A -85,B 0,C 180,E1 -24059.452,E2 -24059.452} C_VEL
LIN {X 0,Y 175.275,Z 446.97,A -85,B 0,C 180,E1 -24061.037,E2 -24061.037} C_VEL
LIN {X 0,Y 168.549,Z 432.824,A -85,B 0,C 180,E1 -24063.493,E2 -24063.493} C_VEL
LIN {X 0,Y 162.315,Z 421.868,A -85,B 0,C 180,E1 -24065.909,E2 -24065.909} C_VEL
LIN {X 0,Y 157.742,Z 414.854,A -85,B 0,C 180,E1 -24067.805,E2 -24067.805} C_VEL
LIN {X 0,Y 155.494,Z 411.48,A -85,B 0,C 180,E1 -24068.795,E2 -24068.795} C_VEL
LIN {X 0,Y 153.376,Z 408.211,A -85,B 0,C 180,E1 -24069.777,E2 -24069.777} C_VEL
LIN {X 0,Y 152.485,Z 407.126,A -85,B 0,C 180,E1 -24070.184,E2 -24070.184} C_VEL
LIN {X 0,Y 150.759,Z 404.853,A -85,B 0,C 180,E1 -24071.006,E2 -24071.006} C_VEL
LIN {X 0,Y 150.172,Z 402.762,A -85,B 0,C 180,E1 -24071.424,E2 -24071.424} C_VEL
LIN {X 0,Y 150.176,Z 402.766,A -85,B 0,C 180,E1 -24075.413,E2 -24075.413} C_VEL
LIN {X 0,Y 150.222,Z 402.756,A -85,B 0,C 180,E1 -24079.081,E2 -24079.081} C_VEL
LIN {X 0,Y 150.238,Z 402.761,A -85,B 0,C 180,E1 -24082.676,E2 -24082.676} C_VEL
LIN {X 0,Y 150.216,Z 402.758,A -85,B 0,C 180,E1 -24087.365,E2 -24087.365} C_VEL
LIN {X 0,Y 150.242,Z 402.748,A -85,B 0,C 180,E1 -24092.717,E2 -24092.717} C_VEL
LIN {X 0,Y 150.388,Z 402.751,A -85,B 0,C 180,E1 -24099.168,E2 -24099.168} C_VEL
LIN {X 0,Y 150.372,Z 402.722,A -85,B 0,C 180,E1 -24103.714,E2 -24103.714} C_VEL
LIN {X 0,Y 150.646,Z 402.718,A -85,B 0,C 180,E1 -24109.244,E2 -24109.244} C_VEL
LIN {X 0,Y 150.739,Z 402.695,A -85,B 0,C 180,E1 -24111.959,E2 -24111.959} C_VEL
LIN {X 0,Y 151.216,Z 402.648,A -85,B 0,C 180,E1 -24119.999,E2 -24119.999} C_VEL
LIN {X 0,Y 150.741,Z 402.7,A -85,B 0,C 180,E1 -24128.04,E2 -24128.04} C_VEL
LIN {X 0,Y 150.611,Z 402.725,A -85,B 0,C 180,E1 -24131.506,E2 -24131.506} C_VEL
LIN {X 0,Y 150.393,Z 402.753,A -85,B 0,C 180,E1 -24136.283,E2 -24136.283} C_VEL
LIN {X 0,Y 150.387,Z 402.753,A -85,B 0,C 180,E1 -24140.831,E2 -24140.831} C_VEL
LIN {X 0,Y 150.241,Z 402.768,A -85,B 0,C 180,E1 -24147.282,E2 -24147.282} C_VEL
LIN {X 0,Y 150.214,Z 402.776,A -85,B 0,C 180,E1 -24152.634,E2 -24152.634} C_VEL
LIN {X 0,Y 150.276,Z 402.872,A -85,B 0,C 180,E1 -24158.934,E2 -24158.934} C_VEL
LIN {X 0,Y 151.383,Z 405.848,A -85,B 0,C 180,E1 -24159.668,E2 -24159.668} C_VEL
LIN {X 0,Y 153.888,Z 409.102,A -85,B 0,C 180,E1 -24160.833,E2 -24160.833} C_VEL
LIN {X 0,Y 159.359,Z 418.996,A -85,B 0,C 180,E1 -24163.344,E2 -24163.344} C_VEL
LIN {X 0,Y 165.137,Z 430.757,A -85,B 0,C 180,E1 -24165.794,E2 -24165.794} C_VEL
LIN {X 0,Y 170.408,Z 443.605,A -85,B 0,C 180,E1 -24167.932,E2 -24167.932} C_VEL
LIN {X 0,Y 172.682,Z 450.407,A -85,B 0,C 180,E1 -24168.861,E2 -24168.861} C_VEL
LIN {X 0,Y 174.249,Z 471.568,A -85,B 0,C 180,E1 -24170.304,E2 -24170.304} C_VEL
LIN {X 0,Y 171.811,Z 513.652,A -85,B 0,C 180,E1 -24171.926,E2 -24171.926} C_VEL
LIN {X 0,Y 170.205,Z 527.013,A -85,B 0,C 180,E1 -24172.852,E2 -24172.852} C_VEL
LIN {X 0,Y 168.084,Z 539.534,A -85,B 0,C 180,E1 -24174.171,E2 -24174.171} C_VEL
LIN {X 0,Y 165.545,Z 550.669,A -85,B 0,C 180,E1 -24175.771,E2 -24175.771} C_VEL
LIN {X 0,Y 162.816,Z 560.986,A -85,B 0,C 180,E1 -24177.713,E2 -24177.713} C_VEL
LIN {X 0,Y 159.577,Z 571.669,A -85,B 0,C 180,E1 -24180.3,E2 -24180.3} C_VEL
LIN {X 0,Y 156.568,Z 581.313,A -85,B 0,C 180,E1 -24183.329,E2 -24183.329} C_VEL
LIN {X 0,Y 154.027,Z 589.201,A -85,B 0,C 180,E1 -24186.469,E2 -24186.469} C_VEL
LIN {X 0,Y 151.544,Z 596.891,A -85,B 0,C 180,E1 -24190.353,E2 -24190.353} C_VEL
LIN {X 0,Y 149.356,Z 603.978,A -85,B 0,C 180,E1 -24195.001,E2 -24195.001} C_VEL
LIN {X 0,Y 148.389,Z 608.233,A -85,B 0,C 180,E1 -24198.657,E2 -24198.657} C_VEL
LIN {X 0,Y 147.464,Z 610.31,A -85,B 0,C 180,E1 -24200.768,E2 -24200.768} C_VEL
LIN {X 0,Y 145.818,Z 612.055,A -85,B 0,C 180,E1 -24202.89,E2 -24202.89} C_VEL
LIN {X 0,Y 142.148,Z 614.592,A -85,B 0,C 180,E1 -24207.317,E2 -24207.317} C_VEL
LIN {X 0,Y 140.868,Z 615.65,A -85,B 0,C 180,E1 -24210.48,E2 -24210.48} C_VEL
LIN {X 0,Y 140.735,Z 616.251,A -85,B 0,C 180,E1 -24212.862,E2 -24212.862} C_VEL
LIN {X 0,Y 140.675,Z 616.569,A -85,B 0,C 180,E1 -24215.734,E2 -24215.734} C_VEL
LIN {X 0,Y 141.342,Z 616.063,A -85,B 0,C 180,E1 -24221.472,E2 -24221.472} C_VEL
LIN {X 0,Y 142.147,Z 615.212,A -85,B 0,C 180,E1 -24224.312,E2 -24224.312} C_VEL
LIN {X 0,Y 143.232,Z 613.945,A -85,B 0,C 180,E1 -24227.121,E2 -24227.121} C_VEL
LIN {X 0,Y 146.62,Z 610.221,A -85,B 0,C 180,E1 -24232.548,E2 -24232.548} C_VEL
LIN {X 0,Y 150.013,Z 606.235,A -85,B 0,C 180,E1 -24236.427,E2 -24236.427} C_VEL
LIN {X 0,Y 153.859,Z 601.135,A -85,B 0,C 180,E1 -24240.162,E2 -24240.162} C_VEL
LIN {X 0,Y 158.493,Z 594.759,A -85,B 0,C 180,E1 -24243.66,E2 -24243.66} C_VEL
LIN {X 0,Y 163.807,Z 586.813,A -85,B 0,C 180,E1 -24246.916,E2 -24246.916} C_VEL
LIN {X 0,Y 168.653,Z 578.745,A -85,B 0,C 180,E1 -24249.455,E2 -24249.455} C_VEL
LIN {X 0,Y 173.324,Z 569.992,A -85,B 0,C 180,E1 -24251.603,E2 -24251.603} C_VEL
LIN {X 0,Y 178.225,Z 559.306,A -85,B 0,C 180,E1 -24253.635,E2 -24253.635} C_VEL
LIN {X 0,Y 182.278,Z 548.964,A -85,B 0,C 180,E1 -24255.11,E2 -24255.11} C_VEL
LIN {X 0,Y 185.782,Z 537.962,A -85,B 0,C 180,E1 -24256.297,E2 -24256.297} C_VEL
LIN {X 0,Y 188.979,Z 524.459,A -85,B 0,C 180,E1 -24257.346,E2 -24257.346} C_VEL
LIN {X 0,Y 191.125,Z 510.875,A -85,B 0,C 180,E1 -24258.026,E2 -24258.026} C_VEL
LIN {X 0,Y 193.302,Z 481.39,A -85,B 0,C 180,E1 -24259.018,E2 -24259.018} C_VEL
LIN {X 0,Y 189.108,Z 470.514,A -85,B 0,C 180,E1 -24261.433,E2 -24261.433} C_VEL
LIN {X 0,Y 184.893,Z 461.077,A -85,B 0,C 180,E1 -24264.032,E2 -24264.032} C_VEL
LIN {X 0,Y 180.894,Z 452.958,A -85,B 0,C 180,E1 -24266.755,E2 -24266.755} C_VEL
LIN {X 0,Y 177.977,Z 447.589,A -85,B 0,C 180,E1 -24268.936,E2 -24268.936} C_VEL
LIN {X 0,Y 175.542,Z 443.285,A -85,B 0,C 180,E1 -24270.934,E2 -24270.934} C_VEL
LIN {X 0,Y 172.815,Z 438.598,A -85,B 0,C 180,E1 -24273.427,E2 -24273.427} C_VEL
LIN {X 0,Y 169.824,Z 433.664,A -85,B 0,C 180,E1 -24276.588,E2 -24276.588} C_VEL
LIN {X 0,Y 166.075,Z 428.571,A -85,B 0,C 180,E1 -24281.512,E2 -24281.512} C_VEL
LIN {X 0,Y 165.649,Z 427.629,A -85,B 0,C 180,E1 -24282.266,E2 -24282.266} C_VEL
LIN {X 0,Y 162.892,Z 425.253,A -85,B 0,C 180,E1 -24287.806,E2 -24287.806} C_VEL
LIN {X 0,Y 161.94,Z 422.053,A -85,B 0,C 180,E1 -24292.52,E2 -24292.52} C_VEL
LIN {X 0,Y 162.128,Z 422.065,A -85,B 0,C 180,E1 -24300.156,E2 -24300.156} C_VEL
LIN {X 0,Y 162.748,Z 424.658,A -85,B 0,C 180,E1 -24303.327,E2 -24303.327} C_VEL
LIN {X 0,Y 165.929,Z 427.864,A -85,B 0,C 180,E1 -24309.851,E2 -24309.851} C_VEL
LIN {X 0,Y 167.81,Z 431.176,A -85,B 0,C 180,E1 -24312.702,E2 -24312.702} C_VEL
LIN {X 0,Y 169.788,Z 433.071,A -85,B 0,C 180,E1 -24314.994,E2 -24314.994} C_VEL
LIN {X 0,Y 172.31,Z 436.793,A -85,B 0,C 180,E1 -24317.66,E2 -24317.66} C_VEL
LIN {X 0,Y 173.649,Z 438.405,A -85,B 0,C 180,E1 -24318.892,E2 -24318.892} C_VEL
LIN {X 0,Y 176.927,Z 443.069,A -85,B 0,C 180,E1 -24321.673,E2 -24321.673} C_VEL
LIN {X 0,Y 180.078,Z 447.736,A -85,B 0,C 180,E1 -24324.039,E2 -24324.039} C_VEL
LIN {X 0,Y 184.617,Z 454.884,A -85,B 0,C 180,E1 -24327.068,E2 -24327.068} C_VEL
LIN {X 0,Y 189.534,Z 463.22,A -85,B 0,C 180,E1 -24329.963,E2 -24329.963} C_VEL
LIN {X 0,Y 194.041,Z 471.986,A -85,B 0,C 180,E1 -24332.389,E2 -24332.389} C_VEL
LIN {X 0,Y 191.59,Z 501.844,A -85,B 0,C 180,E1 -24333.365,E2 -24333.365} C_VEL
LIN {X 0,Y 189.511,Z 515.112,A -85,B 0,C 180,E1 -24334.136,E2 -24334.136} C_VEL
LIN {X 0,Y 186.697,Z 527.723,A -85,B 0,C 180,E1 -24335.276,E2 -24335.276} C_VEL
LIN {X 0,Y 182.871,Z 539.6,A -85,B 0,C 180,E1 -24336.656,E2 -24336.656} C_VEL
LIN {X 0,Y 178.509,Z 550.898,A -85,B 0,C 180,E1 -24338.469,E2 -24338.469} C_VEL
LIN {X 0,Y 173.912,Z 561.256,A -85,B 0,C 180,E1 -24340.739,E2 -24340.739} C_VEL
LIN {X 0,Y 168.927,Z 570.427,A -85,B 0,C 180,E1 -24343.277,E2 -24343.277} C_VEL
LIN {X 0,Y 163.398,Z 579.329,A -85,B 0,C 180,E1 -24346.515,E2 -24346.515} C_VEL
LIN {X 0,Y 158.433,Z 586.397,A -85,B 0,C 180,E1 -24349.969,E2 -24349.969} C_VEL
LIN {X 0,Y 153.989,Z 592.002,A -85,B 0,C 180,E1 -24353.608,E2 -24353.608} C_VEL
LIN {X 0,Y 150.201,Z 596.32,A -85,B 0,C 180,E1 -24357.379,E2 -24357.379} C_VEL
LIN {X 0,Y 146.937,Z 599.639,A -85,B 0,C 180,E1 -24361.426,E2 -24361.426} C_VEL
LIN {X 0,Y 145.188,Z 601.245,A -85,B 0,C 180,E1 -24364.174,E2 -24364.174} C_VEL
LIN {X 0,Y 142.827,Z 603.072,A -85,B 0,C 180,E1 -24369.219,E2 -24369.219} C_VEL
LIN {X 0,Y 141.731,Z 603.527,A -85,B 0,C 180,E1 -24372.692,E2 -24372.692} C_VEL
LIN {X 0,Y 140.696,Z 603.047,A -85,B 0,C 180,E1 -24378.475,E2 -24378.475} C_VEL
LIN {X 0,Y 140.63,Z 602.174,A -85,B 0,C 180,E1 -24381.378,E2 -24381.378} C_VEL
LIN {X 0,Y 140.996,Z 600.248,A -85,B 0,C 180,E1 -24385.508,E2 -24385.508} C_VEL
LIN {X 0,Y 141.586,Z 597.136,A -85,B 0,C 180,E1 -24390,E2 -24390} C_VEL
LIN {X 0,Y 142.741,Z 593.108,A -85,B 0,C 180,E1 -24394.235,E2 -24394.235} C_VEL
LIN {X 0,Y 144.791,Z 586.925,A -85,B 0,C 180,E1 -24399.076,E2 -24399.076} C_VEL
LIN {X 0,Y 147.194,Z 580.202,A -85,B 0,C 180,E1 -24403.108,E2 -24403.108} C_VEL
LIN {X 0,Y 150.236,Z 571.846,A -85,B 0,C 180,E1 -24407,E2 -24407} C_VEL
LIN {X 0,Y 153.242,Z 563.232,A -85,B 0,C 180,E1 -24410.118,E2 -24410.118} C_VEL
LIN {X 0,Y 156.699,Z 552.617,A -85,B 0,C 180,E1 -24413.106,E2 -24413.106} C_VEL
LIN {X 0,Y 159.609,Z 542.09,A -85,B 0,C 180,E1 -24415.424,E2 -24415.424} C_VEL
LIN {X 0,Y 162.266,Z 530.392,A -85,B 0,C 180,E1 -24417.398,E2 -24417.398} C_VEL
LIN {X 0,Y 164.648,Z 516.956,A -85,B 0,C 180,E1 -24419.047,E2 -24419.047} C_VEL
LIN {X 0,Y 166.24,Z 503.9,A -85,B 0,C 180,E1 -24420.134,E2 -24420.134} C_VEL
LIN {X 0,Y 167.223,Z 490.136,A -85,B 0,C 180,E1 -24420.801,E2 -24420.801} C_VEL
LIN {X 0,Y 169.483,Z 449.117,A -85,B 0,C 180,E1 -24422.377,E2 -24422.377} C_VEL
LIN {X 0,Y 163.326,Z 436.072,A -85,B 0,C 180,E1 -24424.794,E2 -24424.794} C_VEL
LIN {X 0,Y 157.346,Z 425.54,A -85,B 0,C 180,E1 -24427.286,E2 -24427.286} C_VEL
LIN {X 0,Y 151.836,Z 416.944,A -85,B 0,C 180,E1 -24429.783,E2 -24429.783} C_VEL
LIN {X 0,Y 148.701,Z 412.513,A -85,B 0,C 180,E1 -24431.307,E2 -24431.307} C_VEL
LIN {X 0,Y 146.498,Z 409.084,A -85,B 0,C 180,E1 -24432.466,E2 -24432.466} C_VEL
LIN {X 0,Y 143.991,Z 406.343,A -85,B 0,C 180,E1 -24433.774,E2 -24433.774} C_VEL
LIN {X 0,Y 143.127,Z 403.653,A -85,B 0,C 180,E1 -24434.426,E2 -24434.426} C_VEL
LIN {X 0,Y 143.121,Z 403.652,A -85,B 0,C 180,E1 -24440.328,E2 -24440.328} C_VEL
LIN {X 0,Y 143.168,Z 403.627,A -85,B 0,C 180,E1 -24446.564,E2 -24446.564} C_VEL
LIN {X 0,Y 143.189,Z 403.632,A -85,B 0,C 180,E1 -24452.062,E2 -24452.062} C_VEL
LIN {X 0,Y 143.309,Z 403.634,A -85,B 0,C 180,E1 -24458.71,E2 -24458.71} C_VEL
LIN {X 0,Y 143.316,Z 403.604,A -85,B 0,C 180,E1 -24462.888,E2 -24462.888} C_VEL
LIN {X 0,Y 143.592,Z 403.596,A -85,B 0,C 180,E1 -24468.709,E2 -24468.709} C_VEL
LIN {X 0,Y 143.659,Z 403.58,A -85,B 0,C 180,E1 -24471.56,E2 -24471.56} C_VEL
LIN {X 0,Y 144.174,Z 403.525,A -85,B 0,C 180,E1 -24479.999,E2 -24479.999} C_VEL
LIN {X 0,Y 143.662,Z 403.581,A -85,B 0,C 180,E1 -24488.439,E2 -24488.439} C_VEL
LIN {X 0,Y 143.545,Z 403.604,A -85,B 0,C 180,E1 -24491.712,E2 -24491.712} C_VEL
LIN {X 0,Y 143.332,Z 403.631,A -85,B 0,C 180,E1 -24497.109,E2 -24497.109} C_VEL
LIN {X 0,Y 143.308,Z 403.635,A -85,B 0,C 180,E1 -24501.289,E2 -24501.289} C_VEL
LIN {X 0,Y 143.187,Z 403.645,A -85,B 0,C 180,E1 -24507.937,E2 -24507.937} C_VEL
LIN {X 0,Y 143.165,Z 403.654,A -85,B 0,C 180,E1 -24513.435,E2 -24513.435} C_VEL
LIN {X 0,Y 143.147,Z 403.8,A -85,B 0,C 180,E1 -24516.004,E2 -24516.004} C_VEL
LIN {X 0,Y 144.114,Z 406.453,A -85,B 0,C 180,E1 -24516.649,E2 -24516.649} C_VEL
LIN {X 0,Y 146.618,Z 409.209,A -85,B 0,C 180,E1 -24517.954,E2 -24517.954} C_VEL
LIN {X 0,Y 148.763,Z 412.515,A -85,B 0,C 180,E1 -24519.079,E2 -24519.079} C_VEL
LIN {X 0,Y 149.97,Z 414.248,A -85,B 0,C 180,E1 -24519.68,E2 -24519.68} C_VEL
LIN {X 0,Y 154.912,Z 423.411,A -85,B 0,C 180,E1 -24522.111,E2 -24522.111} C_VEL
LIN {X 0,Y 160.553,Z 435.182,A -85,B 0,C 180,E1 -24524.677,E2 -24524.677} C_VEL
LIN {X 0,Y 165.989,Z 448.979,A -85,B 0,C 180,E1 -24527.038,E2 -24527.038} C_VEL
LIN {X 0,Y 167.202,Z 453.151,A -85,B 0,C 180,E1 -24527.593,E2 -24527.593} C_VEL
LIN {X 0,Y 168.496,Z 472.122,A -85,B 0,C 180,E1 -24528.935,E2 -24528.935} C_VEL
LIN {X 0,Y 165.975,Z 513.513,A -85,B 0,C 180,E1 -24530.569,E2 -24530.569} C_VEL
LIN {X 0,Y 164.223,Z 527.235,A -85,B 0,C 180,E1 -24531.548,E2 -24531.548} C_VEL
LIN {X 0,Y 162.139,Z 539.059,A -85,B 0,C 180,E1 -24532.835,E2 -24532.835} C_VEL
LIN {X 0,Y 159.273,Z 551.025,A -85,B 0,C 180,E1 -24534.61,E2 -24534.61} C_VEL
LIN {X 0,Y 156.429,Z 561.216,A -85,B 0,C 180,E1 -24536.609,E2 -24536.609} C_VEL
LIN {X 0,Y 153.059,Z 571.802,A -85,B 0,C 180,E1 -24539.282,E2 -24539.282} C_VEL
LIN {X 0,Y 150.213,Z 580.471,A -85,B 0,C 180,E1 -24542.105,E2 -24542.105} C_VEL
LIN {X 0,Y 147.305,Z 588.843,A -85,B 0,C 180,E1 -24545.529,E2 -24545.529} C_VEL
LIN {X 0,Y 144.816,Z 596.236,A -85,B 0,C 180,E1 -24549.4,E2 -24549.4} C_VEL
LIN {X 0,Y 143.009,Z 601.546,A -85,B 0,C 180,E1 -24552.851,E2 -24552.851} C_VEL
LIN {X 0,Y 141.625,Z 606.692,A -85,B 0,C 180,E1 -24557.097,E2 -24557.097} C_VEL
LIN {X 0,Y 140.913,Z 610.675,A -85,B 0,C 180,E1 -24561.395,E2 -24561.395} C_VEL
LIN {X 0,Y 140.772,Z 614.184,A -85,B 0,C 180,E1 -24566.849,E2 -24566.849} C_VEL
LIN {X 0,Y 140.868,Z 615.65,A -85,B 0,C 180,E1 -24570.48,E2 -24570.48} C_VEL
LIN {X 0,Y 140.01,Z 616.21,A -85,B 0,C 180,E1 -24572.856,E2 -24572.856} C_VEL
LIN {X 0,Y 137.141,Z 616.428,A -85,B 0,C 180,E1 -24576.783,E2 -24576.783} C_VEL
LIN {X 0,Y 135.066,Z 616.15,A -85,B 0,C 180,E1 -24580.032,E2 -24580.032} C_VEL
LIN {X 0,Y 134.597,Z 615.563,A -85,B 0,C 180,E1 -24582.962,E2 -24582.962} C_VEL
LIN {X 0,Y 134.693,Z 615.409,A -85,B 0,C 180,E1 -24583.38,E2 -24583.38} C_VEL
LIN {X 0,Y 136.428,Z 613.712,A -85,B 0,C 180,E1 -24588.004,E2 -24588.004} C_VEL
LIN {X 0,Y 140.052,Z 610.036,A -85,B 0,C 180,E1 -24593.668,E2 -24593.668} C_VEL
LIN {X 0,Y 143.659,Z 606.102,A -85,B 0,C 180,E1 -24597.694,E2 -24597.694} C_VEL
LIN {X 0,Y 147.753,Z 601.057,A -85,B 0,C 180,E1 -24601.548,E2 -24601.548} C_VEL
LIN {X 0,Y 152.62,Z 594.758,A -85,B 0,C 180,E1 -24605.142,E2 -24605.142} C_VEL
LIN {X 0,Y 158.18,Z 586.904,A -85,B 0,C 180,E1 -24608.463,E2 -24608.463} C_VEL
LIN {X 0,Y 164.313,Z 577.14,A -85,B 0,C 180,E1 -24611.525,E2 -24611.525} C_VEL
LIN {X 0,Y 169.234,Z 568.136,A -85,B 0,C 180,E1 -24613.661,E2 -24613.661} C_VEL
LIN {X 0,Y 173.779,Z 558.424,A -85,B 0,C 180,E1 -24615.461,E2 -24615.461} C_VEL
LIN {X 0,Y 177.973,Z 547.924,A -85,B 0,C 180,E1 -24616.931,E2 -24616.931} C_VEL
LIN {X 0,Y 181.826,Z 535.828,A -85,B 0,C 180,E1 -24618.188,E2 -24618.188} C_VEL
LIN {X 0,Y 184.907,Z 522.719,A -85,B 0,C 180,E1 -24619.167,E2 -24619.167} C_VEL
LIN {X 0,Y 186.952,Z 509.462,A -85,B 0,C 180,E1 -24619.787,E2 -24619.787} C_VEL
LIN {X 0,Y 188.893,Z 483.843,A -85,B 0,C 180,E1 -24620.66,E2 -24620.66} C_VEL
LIN {X 0,Y 184.844,Z 473.142,A -85,B 0,C 180,E1 -24623.2,E2 -24623.2} C_VEL
LIN {X 0,Y 180.396,Z 463.033,A -85,B 0,C 180,E1 -24626.234,E2 -24626.234} C_VEL
LIN {X 0,Y 176.373,Z 454.84,A -85,B 0,C 180,E1 -24629.317,E2 -24629.317} C_VEL
LIN {X 0,Y 173.06,Z 448.879,A -85,B 0,C 180,E1 -24632.175,E2 -24632.175} C_VEL
LIN {X 0,Y 170.882,Z 444.882,A -85,B 0,C 180,E1 -24634.321,E2 -24634.321} C_VEL
LIN {X 0,Y 168.009,Z 440.004,A -85,B 0,C 180,E1 -24637.561,E2 -24637.561} C_VEL
LIN {X 0,Y 164.626,Z 435.052,A -85,B 0,C 180,E1 -24642.383,E2 -24642.383} C_VEL
LIN {X 0,Y 164.345,Z 434.489,A -85,B 0,C 180,E1 -24642.903,E2 -24642.903} C_VEL
LIN {X 0,Y 161.795,Z 432.035,A -85,B 0,C 180,E1 -24648.458,E2 -24648.458} C_VEL
LIN {X 0,Y 161.06,Z 429.236,A -85,B 0,C 180,E1 -24652.479,E2 -24652.479} C_VEL
LIN {X 0,Y 161.162,Z 429.013,A -85,B 0,C 180,E1 -24659.632,E2 -24659.632} C_VEL
LIN {X 0,Y 161.792,Z 431.709,A -85,B 0,C 180,E1 -24663.114,E2 -24663.114} C_VEL
LIN {X 0,Y 164.573,Z 434.584,A -85,B 0,C 180,E1 -24669.138,E2 -24669.138} C_VEL
LIN {X 0,Y 166.482,Z 437.985,A -85,B 0,C 180,E1 -24672.186,E2 -24672.186} C_VEL
LIN {X 0,Y 168.285,Z 439.916,A -85,B 0,C 180,E1 -24674.396,E2 -24674.396} C_VEL
LIN {X 0,Y 170.847,Z 443.635,A -85,B 0,C 180,E1 -24677.198,E2 -24677.198} C_VEL
LIN {X 0,Y 172.169,Z 445.509,A -85,B 0,C 180,E1 -24678.482,E2 -24678.482} C_VEL
LIN {X 0,Y 174.979,Z 449.607,A -85,B 0,C 180,E1 -24680.961,E2 -24680.961} C_VEL
LIN {X 0,Y 178.947,Z 455.66,A -85,B 0,C 180,E1 -24684.028,E2 -24684.028} C_VEL
LIN {X 0,Y 184.884,Z 465.73,A -85,B 0,C 180,E1 -24687.985,E2 -24687.985} C_VEL
LIN {X 0,Y 189.632,Z 474.971,A -85,B 0,C 180,E1 -24690.771,E2 -24690.771} C_VEL
LIN {X 0,Y 187.295,Z 502.172,A -85,B 0,C 180,E1 -24691.664,E2 -24691.664} C_VEL
LIN {X 0,Y 185.064,Z 515.85,A -85,B 0,C 180,E1 -24692.463,E2 -24692.463} C_VEL
LIN {X 0,Y 182.316,Z 527.685,A -85,B 0,C 180,E1 -24693.531,E2 -24693.531} C_VEL
LIN {X 0,Y 178.676,Z 538.843,A -85,B 0,C 180,E1 -24694.808,E2 -24694.808} C_VEL
LIN {X 0,Y 174.61,Z 549.154,A -85,B 0,C 180,E1 -24696.392,E2 -24696.392} C_VEL
LIN {X 0,Y 169.815,Z 559.831,A -85,B 0,C 180,E1 -24698.634,E2 -24698.634} C_VEL
LIN {X 0,Y 165.063,Z 568.497,A -85,B 0,C 180,E1 -24700.91,E2 -24700.91} C_VEL
LIN {X 0,Y 160.086,Z 576.443,A -85,B 0,C 180,E1 -24703.585,E2 -24703.585} C_VEL
LIN {X 0,Y 154.624,Z 584.146,A -85,B 0,C 180,E1 -24707.018,E2 -24707.018} C_VEL
LIN {X 0,Y 149.723,Z 590.294,A -85,B 0,C 180,E1 -24710.678,E2 -24710.678} C_VEL
LIN {X 0,Y 145.406,Z 595.134,A -85,B 0,C 180,E1 -24714.55,E2 -24714.55} C_VEL
LIN {X 0,Y 141.699,Z 598.82,A -85,B 0,C 180,E1 -24718.616,E2 -24718.616} C_VEL
LIN {X 0,Y 138.696,Z 601.457,A -85,B 0,C 180,E1 -24722.868,E2 -24722.868} C_VEL
LIN {X 0,Y 135.922,Z 603.444,A -85,B 0,C 180,E1 -24728.548,E2 -24728.548} C_VEL
LIN {X 0,Y 134.838,Z 603.853,A -85,B 0,C 180,E1 -24731.777,E2 -24731.777} C_VEL
LIN {X 0,Y 133.659,Z 603.427,A -85,B 0,C 180,E1 -24737.859,E2 -24737.859} C_VEL
LIN {X 0,Y 133.527,Z 602.611,A -85,B 0,C 180,E1 -24740.915,E2 -24740.915} C_VEL
LIN {X 0,Y 133.922,Z 600.519,A -85,B 0,C 180,E1 -24745.642,E2 -24745.642} C_VEL
LIN {X 0,Y 134.496,Z 597.668,A -85,B 0,C 180,E1 -24750,E2 -24750} C_VEL
LIN {X 0,Y 135.662,Z 593.703,A -85,B 0,C 180,E1 -24754.457,E2 -24754.457} C_VEL
LIN {X 0,Y 137.784,Z 587.608,A -85,B 0,C 180,E1 -24759.542,E2 -24759.542} C_VEL
LIN {X 0,Y 140.303,Z 580.96,A -85,B 0,C 180,E1 -24763.764,E2 -24763.764} C_VEL
LIN {X 0,Y 143.493,Z 572.712,A -85,B 0,C 180,E1 -24767.825,E2 -24767.825} C_VEL
LIN {X 0,Y 146.613,Z 564.239,A -85,B 0,C 180,E1 -24771.07,E2 -24771.07} C_VEL
LIN {X 0,Y 150.218,Z 553.762,A -85,B 0,C 180,E1 -24774.165,E2 -24774.165} C_VEL
LIN {X 0,Y 153.668,Z 541.979,A -85,B 0,C 180,E1 -24776.848,E2 -24776.848} C_VEL
LIN {X 0,Y 156.467,Z 530.118,A -85,B 0,C 180,E1 -24778.871,E2 -24778.871} C_VEL
LIN {X 0,Y 158.751,Z 517.787,A -85,B 0,C 180,E1 -24780.42,E2 -24780.42} C_VEL
LIN {X 0,Y 160.417,Z 505.075,A -85,B 0,C 180,E1 -24781.532,E2 -24781.532} C_VEL
LIN {X 0,Y 161.479,Z 491.257,A -85,B 0,C 180,E1 -24782.239,E2 -24782.239} C_VEL
LIN {X 0,Y 163.872,Z 452.049,A -85,B 0,C 180,E1 -24783.742,E2 -24783.742} C_VEL
LIN {X 0,Y 162.909,Z 449.271,A -85,B 0,C 180,E1 -24784.172,E2 -24784.172} C_VEL
LIN {X 0,Y 157.531,Z 438.099,A -85,B 0,C 180,E1 -24786.466,E2 -24786.466} C_VEL
LIN {X 0,Y 150.741,Z 426.311,A -85,B 0,C 180,E1 -24789.578,E2 -24789.578} C_VEL
LIN {X 0,Y 144.831,Z 417.587,A -85,B 0,C 180,E1 -24792.573,E2 -24792.573} C_VEL
LIN {X 0,Y 142.352,Z 414.032,A -85,B 0,C 180,E1 -24793.95,E2 -24793.95} C_VEL
LIN {X 0,Y 140.085,Z 410.982,A -85,B 0,C 180,E1 -24795.27,E2 -24795.27} C_VEL
LIN {X 0,Y 139.328,Z 409.645,A -85,B 0,C 180,E1 -24795.755,E2 -24795.755} C_VEL
LIN {X 0,Y 137.169,Z 407.472,A -85,B 0,C 180,E1 -24797.058,E2 -24797.058} C_VEL
LIN {X 0,Y 136.131,Z 404.914,A -85,B 0,C 180,E1 -24797.843,E2 -24797.843} C_VEL
LIN {X 0,Y 136.065,Z 404.511,A -85,B 0,C 180,E1 -24798.023,E2 -24798.023} C_VEL
LIN {X 0,Y 136.091,Z 404.53,A -85,B 0,C 180,E1 -24801.704,E2 -24801.704} C_VEL
LIN {X 0,Y 136.092,Z 404.503,A -85,B 0,C 180,E1 -24805.715,E2 -24805.715} C_VEL
LIN {X 0,Y 136.145,Z 404.505,A -85,B 0,C 180,E1 -24812.315,E2 -24812.315} C_VEL
LIN {X 0,Y 136.276,Z 404.51,A -85,B 0,C 180,E1 -24818.837,E2 -24818.837} C_VEL
LIN {X 0,Y 136.277,Z 404.474,A -85,B 0,C 180,E1 -24825.056,E2 -24825.056} C_VEL
LIN {X 0,Y 136.495,Z 404.475,A -85,B 0,C 180,E1 -24828.114,E2 -24828.114} C_VEL
LIN {X 0,Y 136.586,Z 404.464,A -85,B 0,C 180,E1 -24831.119,E2 -24831.119} C_VEL
LIN {X 0,Y 137.131,Z 404.402,A -85,B 0,C 180,E1 -24839.999,E2 -24839.999} C_VEL
LIN {X 0,Y 136.589,Z 404.462,A -85,B 0,C 180,E1 -24848.879,E2 -24848.879} C_VEL
LIN {X 0,Y 136.489,Z 404.482,A -85,B 0,C 180,E1 -24851.954,E2 -24851.954} C_VEL
LIN {X 0,Y 136.271,Z 404.504,A -85,B 0,C 180,E1 -24858.025,E2 -24858.025} C_VEL
LIN {X 0,Y 136.224,Z 404.517,A -85,B 0,C 180,E1 -24861.779,E2 -24861.779} C_VEL
LIN {X 0,Y 136.097,Z 404.528,A -85,B 0,C 180,E1 -24868.616,E2 -24868.616} C_VEL
LIN {X 0,Y 136.143,Z 404.537,A -85,B 0,C 180,E1 -24872.492,E2 -24872.492} C_VEL
LIN {X 0,Y 137.073,Z 407.292,A -85,B 0,C 180,E1 -24873.236,E2 -24873.236} C_VEL
LIN {X 0,Y 139.182,Z 409.555,A -85,B 0,C 180,E1 -24874.524,E2 -24874.524} C_VEL
LIN {X 0,Y 139.74,Z 410.122,A -85,B 0,C 180,E1 -24874.85,E2 -24874.85} C_VEL
LIN {X 0,Y 141.743,Z 413.321,A -85,B 0,C 180,E1 -24876.071,E2 -24876.071} C_VEL
LIN {X 0,Y 143.173,Z 414.945,A -85,B 0,C 180,E1 -24876.854,E2 -24876.854} C_VEL
LIN {X 0,Y 146.232,Z 419.636,A -85,B 0,C 180,E1 -24878.532,E2 -24878.532} C_VEL
LIN {X 0,Y 150.942,Z 428.644,A -85,B 0,C 180,E1 -24881.011,E2 -24881.011} C_VEL
LIN {X 0,Y 156.167,Z 439.938,A -85,B 0,C 180,E1 -24883.559,E2 -24883.559} C_VEL
LIN {X 0,Y 161.044,Z 452.871,A -85,B 0,C 180,E1 -24885.843,E2 -24885.843} C_VEL
LIN {X 0,Y 161.768,Z 455.872,A -85,B 0,C 180,E1 -24886.226,E2 -24886.226} C_VEL
LIN {X 0,Y 162.786,Z 473.067,A -85,B 0,C 180,E1 -24887.474,E2 -24887.474} C_VEL
LIN {X 0,Y 160.287,Z 512.869,A -85,B 0,C 180,E1 -24889.085,E2 -24889.085} C_VEL
LIN {X 0,Y 158.464,Z 526.695,A -85,B 0,C 180,E1 -24890.082,E2 -24890.082} C_VEL
LIN {X 0,Y 156.281,Z 538.579,A -85,B 0,C 180,E1 -24891.395,E2 -24891.395} C_VEL
LIN {X 0,Y 153.537,Z 549.792,A -85,B 0,C 180,E1 -24893.075,E2 -24893.075} C_VEL
LIN {X 0,Y 150.105,Z 561.446,A -85,B 0,C 180,E1 -24895.411,E2 -24895.411} C_VEL
LIN {X 0,Y 146.592,Z 571.936,A -85,B 0,C 180,E1 -24898.173,E2 -24898.173} C_VEL
LIN {X 0,Y 143.297,Z 581.377,A -85,B 0,C 180,E1 -24901.434,E2 -24901.434} C_VEL
LIN {X 0,Y 140.782,Z 587.832,A -85,B 0,C 180,E1 -24904.184,E2 -24904.184} C_VEL
LIN {X 0,Y 139.017,Z 593.125,A -85,B 0,C 180,E1 -24906.934,E2 -24906.934} C_VEL
LIN {X 0,Y 136.589,Z 599.924,A -85,B 0,C 180,E1 -24911.242,E2 -24911.242} C_VEL
LIN {X 0,Y 134.665,Z 606.15,A -85,B 0,C 180,E1 -24916.418,E2 -24916.418} C_VEL
LIN {X 0,Y 133.864,Z 610.185,A -85,B 0,C 180,E1 -24920.938,E2 -24920.938} C_VEL
LIN {X 0,Y 133.631,Z 612.252,A -85,B 0,C 180,E1 -24923.962,E2 -24923.962} C_VEL
LIN {X 0,Y 133.683,Z 614.029,A -85,B 0,C 180,E1 -24927.265,E2 -24927.265} C_VEL
LIN {X 0,Y 133.787,Z 615.216,A -85,B 0,C 180,E1 -24930.368,E2 -24930.368} C_VEL
LIN {X 0,Y 133.635,Z 615.882,A -85,B 0,C 180,E1 -24933.015,E2 -24933.015} C_VEL
LIN {X 0,Y 133.606,Z 616.224,A -85,B 0,C 180,E1 -24936.039,E2 -24936.039} C_VEL
LIN {X 0,Y 134.352,Z 615.761,A -85,B 0,C 180,E1 -24942.078,E2 -24942.078} C_VEL
LIN {X 0,Y 134.693,Z 615.409,A -85,B 0,C 180,E1 -24943.38,E2 -24943.38} C_VEL
LIN {X 0,Y 134.863,Z 614.652,A -85,B 0,C 180,E1 -24945.873,E2 -24945.873} C_VEL
LIN {X 0,Y 133.895,Z 612.855,A -85,B 0,C 180,E1 -24950.021,E2 -24950.021} C_VEL
LIN {X 0,Y 133.644,Z 610.393,A -85,B 0,C 180,E1 -24954.136,E2 -24954.136} C_VEL
LIN {X 0,Y 134.896,Z 608.535,A -85,B 0,C 180,E1 -24956.466,E2 -24956.466} C_VEL
LIN {X 0,Y 139.196,Z 603.905,A -85,B 0,C 180,E1 -24960.872,E2 -24960.872} C_VEL
LIN {X 0,Y 144.183,Z 598.034,A -85,B 0,C 180,E1 -24964.94,E2 -24964.94} C_VEL
LIN {X 0,Y 149.717,Z 591.092,A -85,B 0,C 180,E1 -24968.46,E2 -24968.46} C_VEL
LIN {X 0,Y 155.816,Z 582.424,A -85,B 0,C 180,E1 -24971.703,E2 -24971.703} C_VEL
LIN {X 0,Y 161.214,Z 573.572,A -85,B 0,C 180,E1 -24974.226,E2 -24974.226} C_VEL
LIN {X 0,Y 167.084,Z 562.686,A -85,B 0,C 180,E1 -24976.516,E2 -24976.516} C_VEL
LIN {X 0,Y 171.93,Z 551.71,A -85,B 0,C 180,E1 -24978.244,E2 -24978.244} C_VEL
LIN {X 0,Y 176.353,Z 539.559,A -85,B 0,C 180,E1 -24979.622,E2 -24979.622} C_VEL
LIN {X 0,Y 179.588,Z 527.729,A -85,B 0,C 180,E1 -24980.627,E2 -24980.627} C_VEL
LIN {X 0,Y 182.098,Z 514.76,A -85,B 0,C 180,E1 -24981.363,E2 -24981.363} C_VEL
LIN {X 0,Y 183.792,Z 498.19,A -85,B 0,C 180,E1 -24981.957,E2 -24981.957} C_VEL
LIN {X 0,Y 184.679,Z 486.518,A -85,B 0,C 180,E1 -24982.349,E2 -24982.349} C_VEL
LIN {X 0,Y 181.161,Z 476.974,A -85,B 0,C 180,E1 -24984.754,E2 -24984.754} C_VEL
LIN {X 0,Y 177.259,Z 467.739,A -85,B 0,C 180,E1 -24987.655,E2 -24987.655} C_VEL
LIN {X 0,Y 173.545,Z 459.907,A -85,B 0,C 180,E1 -24990.746,E2 -24990.746} C_VEL
LIN {X 0,Y 170.767,Z 454.636,A -85,B 0,C 180,E1 -24993.35,E2 -24993.35} C_VEL
LIN {X 0,Y 168.763,Z 450.831,A -85,B 0,C 180,E1 -24995.481,E2 -24995.481} C_VEL
LIN {X 0,Y 166.255,Z 446.322,A -85,B 0,C 180,E1 -24998.544,E2 -24998.544} C_VEL
LIN {X 0,Y 163.292,Z 441.73,A -85,B 0,C 180,E1 -25003.112,E2 -25003.112} C_VEL
LIN {X 0,Y 160.432,Z 438.038,A -85,B 0,C 180,E1 -25010.386,E2 -25010.386} C_VEL
LIN {X 0,Y 160.111,Z 436.185,A -85,B 0,C 180,E1 -25013.068,E2 -25013.068} C_VEL
LIN {X 0,Y 160.217,Z 436.05,A -85,B 0,C 180,E1 -25019.214,E2 -25019.214} C_VEL
LIN {X 0,Y 160.818,Z 438.698,A -85,B 0,C 180,E1 -25022.819,E2 -25022.819} C_VEL
LIN {X 0,Y 163.349,Z 441.533,A -85,B 0,C 180,E1 -25028.623,E2 -25028.623} C_VEL
LIN {X 0,Y 165.274,Z 444.913,A -85,B 0,C 180,E1 -25031.809,E2 -25031.809} C_VEL
LIN {X 0,Y 166.664,Z 446.467,A -85,B 0,C 180,E1 -25033.605,E2 -25033.605} C_VEL
LIN {X 0,Y 169.397,Z 450.461,A -85,B 0,C 180,E1 -25036.728,E2 -25036.728} C_VEL
LIN {X 0,Y 172.934,Z 455.928,A -85,B 0,C 180,E1 -25040.122,E2 -25040.122} C_VEL
LIN {X 0,Y 176.538,Z 461.657,A -85,B 0,C 180,E1 -25043.072,E2 -25043.072} C_VEL
LIN {X 0,Y 181.956,Z 471.215,A -85,B 0,C 180,E1 -25046.914,E2 -25046.914} C_VEL
LIN {X 0,Y 185.362,Z 478.034,A -85,B 0,C 180,E1 -25049.073,E2 -25049.073} C_VEL
LIN {X 0,Y 183.17,Z 502.482,A -85,B 0,C 180,E1 -25049.882,E2 -25049.882} C_VEL
LIN {X 0,Y 180.951,Z 515.694,A -85,B 0,C 180,E1 -25050.642,E2 -25050.642} C_VEL
LIN {X 0,Y 177.814,Z 528.666,A -85,B 0,C 180,E1 -25051.815,E2 -25051.815} C_VEL
LIN {X 0,Y 173.413,Z 541.289,A -85,B 0,C 180,E1 -25053.295,E2 -25053.295} C_VEL
LIN {X 0,Y 168.503,Z 552.872,A -85,B 0,C 180,E1 -25055.22,E2 -25055.22} C_VEL
LIN {X 0,Y 163.668,Z 562.628,A -85,B 0,C 180,E1 -25057.442,E2 -25057.442} C_VEL
LIN {X 0,Y 158.29,Z 571.618,A -85,B 0,C 180,E1 -25060.015,E2 -25060.015} C_VEL
LIN {X 0,Y 153.2,Z 579.062,A -85,B 0,C 180,E1 -25062.779,E2 -25062.779} C_VEL
LIN {X 0,Y 147.614,Z 586.347,A -85,B 0,C 180,E1 -25066.343,E2 -25066.343} C_VEL
LIN {X 0,Y 142.569,Z 592.116,A -85,B 0,C 180,E1 -25070.147,E2 -25070.147} C_VEL
LIN {X 0,Y 137.422,Z 597.264,A -85,B 0,C 180,E1 -25074.914,E2 -25074.914} C_VEL
LIN {X 0,Y 134.386,Z 600.005,A -85,B 0,C 180,E1 -25078.469,E2 -25078.469} C_VEL
LIN {X 0,Y 132.281,Z 601.67,A -85,B 0,C 180,E1 -25081.435,E2 -25081.435} C_VEL
LIN {X 0,Y 129.126,Z 603.771,A -85,B 0,C 180,E1 -25087.605,E2 -25087.605} C_VEL
LIN {X 0,Y 127.982,Z 604.178,A -85,B 0,C 180,E1 -25090.763,E2 -25090.763} C_VEL
LIN {X 0,Y 126.63,Z 603.807,A -85,B 0,C 180,E1 -25097.174,E2 -25097.174} C_VEL
LIN {X 0,Y 126.454,Z 603.037,A -85,B 0,C 180,E1 -25100.402,E2 -25100.402} C_VEL
LIN {X 0,Y 126.849,Z 600.788,A -85,B 0,C 180,E1 -25105.789,E2 -25105.789} C_VEL
LIN {X 0,Y 127.675,Z 596.994,A -85,B 0,C 180,E1 -25111.577,E2 -25111.577} C_VEL
LIN {X 0,Y 129.156,Z 592.722,A -85,B 0,C 180,E1 -25116.248,E2 -25116.248} C_VEL
LIN {X 0,Y 131.64,Z 586.275,A -85,B 0,C 180,E1 -25121.549,E2 -25121.549} C_VEL
LIN {X 0,Y 134.473,Z 579.206,A -85,B 0,C 180,E1 -25125.925,E2 -25125.925} C_VEL
LIN {X 0,Y 138.028,Z 570.393,A -85,B 0,C 180,E1 -25130.101,E2 -25130.101} C_VEL
LIN {X 0,Y 141.515,Z 561.35,A -85,B 0,C 180,E1 -25133.409,E2 -25133.409} C_VEL
LIN {X 0,Y 145.003,Z 551.356,A -85,B 0,C 180,E1 -25136.248,E2 -25136.248} C_VEL
LIN {X 0,Y 148.23,Z 540.271,A -85,B 0,C 180,E1 -25138.688,E2 -25138.688} C_VEL
LIN {X 0,Y 151.208,Z 527.861,A -85,B 0,C 180,E1 -25140.748,E2 -25140.748} C_VEL
LIN {X 0,Y 153.512,Z 515.208,A -85,B 0,C 180,E1 -25142.251,E2 -25142.251} C_VEL
LIN {X 0,Y 155.128,Z 501.64,A -85,B 0,C 180,E1 -25143.333,E2 -25143.333} C_VEL
LIN {X 0,Y 157.462,Z 466.384,A -85,B 0,C 180,E1 -25144.81,E2 -25144.81} C_VEL
LIN {X 0,Y 158.135,Z 453.31,A -85,B 0,C 180,E1 -25145.37,E2 -25145.37} C_VEL
LIN {X 0,Y 152.926,Z 442.217,A -85,B 0,C 180,E1 -25147.759,E2 -25147.759} C_VEL
LIN {X 0,Y 146.612,Z 431.103,A -85,B 0,C 180,E1 -25150.867,E2 -25150.867} C_VEL
LIN {X 0,Y 140.834,Z 422.326,A -85,B 0,C 180,E1 -25154.026,E2 -25154.026} C_VEL
LIN {X 0,Y 138.829,Z 419.478,A -85,B 0,C 180,E1 -25155.218,E2 -25155.218} C_VEL
LIN {X 0,Y 135.863,Z 415.278,A -85,B 0,C 180,E1 -25157.105,E2 -25157.105} C_VEL
LIN {X 0,Y 133.596,Z 412.381,A -85,B 0,C 180,E1 -25158.633,E2 -25158.633} C_VEL
LIN {X 0,Y 132.699,Z 410.754,A -85,B 0,C 180,E1 -25159.312,E2 -25159.312} C_VEL
LIN {X 0,Y 130.472,Z 408.876,A -85,B 0,C 180,E1 -25160.88,E2 -25160.88} C_VEL
LIN {X 0,Y 129.261,Z 406.515,A -85,B 0,C 180,E1 -25161.918,E2 -25161.918} C_VEL
LIN {X 0,Y 129.027,Z 405.404,A -85,B 0,C 180,E1 -25162.27,E2 -25162.27} C_VEL
LIN {X 0,Y 128.996,Z 405.393,A -85,B 0,C 180,E1 -25166.986,E2 -25166.986} C_VEL
LIN {X 0,Y 129.033,Z 405.409,A -85,B 0,C 180,E1 -25170.645,E2 -25170.645} C_VEL
LIN {X 0,Y 129.129,Z 405.391,A -85,B 0,C 180,E1 -25177.702,E2 -25177.702} C_VEL
LIN {X 0,Y 129.177,Z 405.384,A -85,B 0,C 180,E1 -25180.946,E2 -25180.946} C_VEL
LIN {X 0,Y 129.414,Z 405.353,A -85,B 0,C 180,E1 -25187.819,E2 -25187.819} C_VEL
LIN {X 0,Y 129.513,Z 405.349,A -85,B 0,C 180,E1 -25190.63,E2 -25190.63} C_VEL
LIN {X 0,Y 130.086,Z 405.279,A -85,B 0,C 180,E1 -25199.999,E2 -25199.999} C_VEL
LIN {X 0,Y 129.515,Z 405.345,A -85,B 0,C 180,E1 -25209.368,E2 -25209.368} C_VEL
LIN {X 0,Y 129.392,Z 405.362,A -85,B 0,C 180,E1 -25212.548,E2 -25212.548} C_VEL
LIN {X 0,Y 129.182,Z 405.385,A -85,B 0,C 180,E1 -25219.051,E2 -25219.051} C_VEL
LIN {X 0,Y 129.133,Z 405.397,A -85,B 0,C 180,E1 -25222.393,E2 -25222.393} C_VEL
LIN {X 0,Y 129.1,Z 405.477,A -85,B 0,C 180,E1 -25228.224,E2 -25228.224} C_VEL
LIN {X 0,Y 129.88,Z 407.989,A -85,B 0,C 180,E1 -25229.003,E2 -25229.003} C_VEL
LIN {X 0,Y 131.784,Z 410.214,A -85,B 0,C 180,E1 -25230.439,E2 -25230.439} C_VEL
LIN {X 0,Y 133.078,Z 411.269,A -85,B 0,C 180,E1 -25231.322,E2 -25231.322} C_VEL
LIN {X 0,Y 135.153,Z 414.564,A -85,B 0,C 180,E1 -25232.805,E2 -25232.805} C_VEL
LIN {X 0,Y 136.58,Z 416.099,A -85,B 0,C 180,E1 -25233.71,E2 -25233.71} C_VEL
LIN {X 0,Y 139.113,Z 419.659,A -85,B 0,C 180,E1 -25235.297,E2 -25235.297} C_VEL
LIN {X 0,Y 142.491,Z 424.817,A -85,B 0,C 180,E1 -25237.282,E2 -25237.282} C_VEL
LIN {X 0,Y 147.861,Z 435.507,A -85,B 0,C 180,E1 -25240.292,E2 -25240.292} C_VEL
LIN {X 0,Y 152.548,Z 446.482,A -85,B 0,C 180,E1 -25242.738,E2 -25242.738} C_VEL
LIN {X 0,Y 156.346,Z 457.4,A -85,B 0,C 180,E1 -25244.67,E2 -25244.67} C_VEL
LIN {X 0,Y 157.247,Z 472.929,A -85,B 0,C 180,E1 -25245.865,E2 -25245.865} C_VEL
LIN {X 0,Y 154.703,Z 512.213,A -85,B 0,C 180,E1 -25247.488,E2 -25247.488} C_VEL
LIN {X 0,Y 152.805,Z 526.149,A -85,B 0,C 180,E1 -25248.504,E2 -25248.504} C_VEL
LIN {X 0,Y 150.545,Z 538.101,A -85,B 0,C 180,E1 -25249.849,E2 -25249.849} C_VEL
LIN {X 0,Y 147.414,Z 550.144,A -85,B 0,C 180,E1 -25251.701,E2 -25251.701} C_VEL
LIN {X 0,Y 144.319,Z 560.378,A -85,B 0,C 180,E1 -25253.811,E2 -25253.811} C_VEL
LIN {X 0,Y 140.613,Z 570.995,A -85,B 0,C 180,E1 -25256.648,E2 -25256.648} C_VEL
LIN {X 0,Y 137.063,Z 580.571,A -85,B 0,C 180,E1 -25260.005,E2 -25260.005} C_VEL
LIN {X 0,Y 134.039,Z 587.921,A -85,B 0,C 180,E1 -25263.26,E2 -25263.26} C_VEL
LIN {X 0,Y 132.494,Z 592.44,A -85,B 0,C 180,E1 -25265.727,E2 -25265.727} C_VEL
LIN {X 0,Y 129.861,Z 599.302,A -85,B 0,C 180,E1 -25270.23,E2 -25270.23} C_VEL
LIN {X 0,Y 127.714,Z 605.594,A -85,B 0,C 180,E1 -25275.663,E2 -25275.663} C_VEL
LIN {X 0,Y 126.841,Z 609.686,A -85,B 0,C 180,E1 -25280.432,E2 -25280.432} C_VEL
LIN {X 0,Y 126.556,Z 611.791,A -85,B 0,C 180,E1 -25283.623,E2 -25283.623} C_VEL
LIN {X 0,Y 126.606,Z 613.857,A -85,B 0,C 180,E1 -25287.693,E2 -25287.693} C_VEL
LIN {X 0,Y 126.74,Z 614.705,A -85,B 0,C 180,E1 -25290,E2 -25290} C_VEL
LIN {X 0,Y 126.547,Z 615.51,A -85,B 0,C 180,E1 -25293.184,E2 -25293.184} C_VEL
LIN {X 0,Y 126.534,Z 615.877,A -85,B 0,C 180,E1 -25296.378,E2 -25296.378} C_VEL
LIN {X 0,Y 127.389,Z 615.46,A -85,B 0,C 180,E1 -25302.749,E2 -25302.749} C_VEL
LIN {X 0,Y 128.365,Z 614.684,A -85,B 0,C 180,E1 -25305.887,E2 -25305.887} C_VEL
LIN {X 0,Y 129.664,Z 613.48,A -85,B 0,C 180,E1 -25308.978,E2 -25308.978} C_VEL
LIN {X 0,Y 132.487,Z 610.938,A -85,B 0,C 180,E1 -25313.443,E2 -25313.443} C_VEL
LIN {X 0,Y 134.896,Z 608.535,A -85,B 0,C 180,E1 -25316.466,E2 -25316.466} C_VEL
LIN {X 0,Y 136.319,Z 606.482,A -85,B 0,C 180,E1 -25318.727,E2 -25318.727} C_VEL
LIN {X 0,Y 137.242,Z 602.731,A -85,B 0,C 180,E1 -25322.563,E2 -25322.563} C_VEL
LIN {X 0,Y 138.633,Z 598.392,A -85,B 0,C 180,E1 -25326.223,E2 -25326.223} C_VEL
LIN {X 0,Y 140.701,Z 595.366,A -85,B 0,C 180,E1 -25328.122,E2 -25328.122} C_VEL
LIN {X 0,Y 146.276,Z 588.453,A -85,B 0,C 180,E1 -25331.347,E2 -25331.347} C_VEL
LIN {X 0,Y 152.834,Z 579.283,A -85,B 0,C 180,E1 -25334.527,E2 -25334.527} C_VEL
LIN {X 0,Y 158.095,Z 570.84,A -85,B 0,C 180,E1 -25336.712,E2 -25336.712} C_VEL
LIN {X 0,Y 163.54,Z 560.54,A -85,B 0,C 180,E1 -25338.767,E2 -25338.767} C_VEL
LIN {X 0,Y 168.642,Z 549.128,A -85,B 0,C 180,E1 -25340.439,E2 -25340.439} C_VEL
LIN {X 0,Y 172.478,Z 538.465,A -85,B 0,C 180,E1 -25341.612,E2 -25341.612} C_VEL
LIN {X 0,Y 175.922,Z 526.042,A -85,B 0,C 180,E1 -25342.605,E2 -25342.605} C_VEL
LIN {X 0,Y 178.432,Z 512.818,A -85,B 0,C 180,E1 -25343.299,E2 -25343.299} C_VEL
LIN {X 0,Y 180.511,Z 490.697,A -85,B 0,C 180,E1 -25344.066,E2 -25344.066} C_VEL
LIN {X 0,Y 180.552,Z 488.932,A -85,B 0,C 180,E1 -25344.176,E2 -25344.176} C_VEL
LIN {X 0,Y 176.805,Z 478.682,A -85,B 0,C 180,E1 -25347.015,E2 -25347.015} C_VEL
LIN {X 0,Y 173.039,Z 469.7,A -85,B 0,C 180,E1 -25350.171,E2 -25350.171} C_VEL
LIN {X 0,Y 169.582,Z 462.318,A -85,B 0,C 180,E1 -25353.477,E2 -25353.477} C_VEL
LIN {X 0,Y 166.836,Z 456.968,A -85,B 0,C 180,E1 -25356.528,E2 -25356.528} C_VEL
LIN {X 0,Y 164.562,Z 452.662,A -85,B 0,C 180,E1 -25359.538,E2 -25359.538} C_VEL
LIN {X 0,Y 162,Z 448.423,A -85,B 0,C 180,E1 -25363.824,E2 -25363.824} C_VEL
LIN {X 0,Y 159.473,Z 445.053,A -85,B 0,C 180,E1 -25370.728,E2 -25370.728} C_VEL
LIN {X 0,Y 159.191,Z 443.178,A -85,B 0,C 180,E1 -25373.505,E2 -25373.505} C_VEL
LIN {X 0,Y 159.287,Z 443.164,A -85,B 0,C 180,E1 -25378.893,E2 -25378.893} C_VEL
LIN {X 0,Y 159.933,Z 445.871,A -85,B 0,C 180,E1 -25382.834,E2 -25382.834} C_VEL
LIN {X 0,Y 162.065,Z 448.315,A -85,B 0,C 180,E1 -25387.946,E2 -25387.946} C_VEL
LIN {X 0,Y 164.075,Z 451.835,A -85,B 0,C 180,E1 -25391.427,E2 -25391.427} C_VEL
LIN {X 0,Y 165.158,Z 453.17,A -85,B 0,C 180,E1 -25392.91,E2 -25392.91} C_VEL
LIN {X 0,Y 168.331,Z 458.122,A -85,B 0,C 180,E1 -25396.681,E2 -25396.681} C_VEL
LIN {X 0,Y 171.024,Z 462.379,A -85,B 0,C 180,E1 -25399.35,E2 -25399.35} C_VEL
LIN {X 0,Y 174.809,Z 468.858,A -85,B 0,C 180,E1 -25402.61,E2 -25402.61} C_VEL
LIN {X 0,Y 179.458,Z 477.439,A -85,B 0,C 180,E1 -25406.063,E2 -25406.063} C_VEL
LIN {X 0,Y 181.278,Z 481.183,A -85,B 0,C 180,E1 -25407.306,E2 -25407.306} C_VEL
LIN {X 0,Y 179.167,Z 503.295,A -85,B 0,C 180,E1 -25408.042,E2 -25408.042} C_VEL
LIN {X 0,Y 176.785,Z 516.816,A -85,B 0,C 180,E1 -25408.834,E2 -25408.834} C_VEL
LIN {X 0,Y 173.474,Z 529.649,A -85,B 0,C 180,E1 -25410.009,E2 -25410.009} C_VEL
LIN {X 0,Y 168.92,Z 542.133,A -85,B 0,C 180,E1 -25411.472,E2 -25411.472} C_VEL
LIN {X 0,Y 164.012,Z 553.228,A -85,B 0,C 180,E1 -25413.325,E2 -25413.325} C_VEL
LIN {X 0,Y 159.114,Z 562.735,A -85,B 0,C 180,E1 -25415.491,E2 -25415.491} C_VEL
LIN {X 0,Y 153.73,Z 571.391,A -85,B 0,C 180,E1 -25417.946,E2 -25417.946} C_VEL
LIN {X 0,Y 147.341,Z 580.299,A -85,B 0,C 180,E1 -25421.303,E2 -25421.303} C_VEL
LIN {X 0,Y 141.522,Z 587.375,A -85,B 0,C 180,E1 -25424.957,E2 -25424.957} C_VEL
LIN {X 0,Y 135.43,Z 593.794,A -85,B 0,C 180,E1 -25429.56,E2 -25429.56} C_VEL
LIN {X 0,Y 130.872,Z 597.983,A -85,B 0,C 180,E1 -25433.793,E2 -25433.793} C_VEL
LIN {X 0,Y 128.254,Z 600.184,A -85,B 0,C 180,E1 -25436.773,E2 -25436.773} C_VEL
LIN {X 0,Y 125.949,Z 601.884,A -85,B 0,C 180,E1 -25439.855,E2 -25439.855} C_VEL
LIN {X 0,Y 122.444,Z 604.044,A -85,B 0,C 180,E1 -25446.311,E2 -25446.311} C_VEL
LIN {X 0,Y 121.179,Z 604.504,A -85,B 0,C 180,E1 -25449.637,E2 -25449.637} C_VEL
LIN {X 0,Y 120.252,Z 604.538,A -85,B 0,C 180,E1 -25453.01,E2 -25453.01} C_VEL
LIN {X 0,Y 119.37,Z 603.448,A -85,B 0,C 180,E1 -25459.827,E2 -25459.827} C_VEL
LIN {X 0,Y 119.774,Z 601.045,A -85,B 0,C 180,E1 -25465.973,E2 -25465.973} C_VEL
LIN {X 0,Y 120.59,Z 597.538,A -85,B 0,C 180,E1 -25471.67,E2 -25471.67} C_VEL
LIN {X 0,Y 122.091,Z 593.332,A -85,B 0,C 180,E1 -25476.611,E2 -25476.611} C_VEL
LIN {X 0,Y 124.721,Z 586.951,A -85,B 0,C 180,E1 -25482.199,E2 -25482.199} C_VEL
LIN {X 0,Y 127.678,Z 579.998,A -85,B 0,C 180,E1 -25486.797,E2 -25486.797} C_VEL
LIN {X 0,Y 131.416,Z 571.277,A -85,B 0,C 180,E1 -25491.16,E2 -25491.16} C_VEL
LIN {X 0,Y 135.45,Z 561.372,A -85,B 0,C 180,E1 -25494.933,E2 -25494.933} C_VEL
LIN {X 0,Y 139.128,Z 551.278,A -85,B 0,C 180,E1 -25497.856,E2 -25497.856} C_VEL
LIN {X 0,Y 142.527,Z 540.102,A -85,B 0,C 180,E1 -25500.359,E2 -25500.359} C_VEL
LIN {X 0,Y 145.641,Z 527.565,A -85,B 0,C 180,E1 -25502.468,E2 -25502.468} C_VEL
LIN {X 0,Y 148.052,Z 514.59,A -85,B 0,C 180,E1 -25504.003,E2 -25504.003} C_VEL
LIN {X 0,Y 149.656,Z 501.678,A -85,B 0,C 180,E1 -25505.028,E2 -25505.028} C_VEL
LIN {X 0,Y 152.681,Z 455.691,A -85,B 0,C 180,E1 -25506.997,E2 -25506.997} C_VEL
LIN {X 0,Y 148.224,Z 446.043,A -85,B 0,C 180,E1 -25509.22,E2 -25509.22} C_VEL
LIN {X 0,Y 142.694,Z 436.04,A -85,B 0,C 180,E1 -25512.16,E2 -25512.16} C_VEL
LIN {X 0,Y 136.133,Z 425.697,A -85,B 0,C 180,E1 -25516.087,E2 -25516.087} C_VEL
LIN {X 0,Y 133.382,Z 421.815,A -85,B 0,C 180,E1 -25517.919,E2 -25517.919} C_VEL
LIN {X 0,Y 130.388,Z 417.772,A -85,B 0,C 180,E1 -25520.081,E2 -25520.081} C_VEL
LIN {X 0,Y 129.353,Z 416.526,A -85,B 0,C 180,E1 -25520.865,E2 -25520.865} C_VEL
LIN {X 0,Y 126.964,Z 413.584,A -85,B 0,C 180,E1 -25522.8,E2 -25522.8} C_VEL
LIN {X 0,Y 126.076,Z 411.863,A -85,B 0,C 180,E1 -25523.633,E2 -25523.633} C_VEL
LIN {X 0,Y 123.375,Z 409.727,A -85,B 0,C 180,E1 -25526.014,E2 -25526.014} C_VEL
LIN {X 0,Y 122.083,Z 407.104,A -85,B 0,C 180,E1 -25527.458,E2 -25527.458} C_VEL
LIN {X 0,Y 121.944,Z 406.278,A -85,B 0,C 180,E1 -25527.783,E2 -25527.783} C_VEL
LIN {X 0,Y 121.951,Z 406.267,A -85,B 0,C 180,E1 -25532.545,E2 -25532.545} C_VEL
LIN {X 0,Y 122.043,Z 406.265,A -85,B 0,C 180,E1 -25537.125,E2 -25537.125} C_VEL
LIN {X 0,Y 122.121,Z 406.237,A -85,B 0,C 180,E1 -25543.276,E2 -25543.276} C_VEL
LIN {X 0,Y 122.361,Z 406.226,A -85,B 0,C 180,E1 -25547.526,E2 -25547.526} C_VEL
LIN {X 0,Y 122.443,Z 406.231,A -85,B 0,C 180,E1 -25550.084,E2 -25550.084} C_VEL
LIN {X 0,Y 122.6,Z 406.178,A -85,B 0,C 180,E1 -25556.713,E2 -25556.713} C_VEL
LIN {X 0,Y 123.04,Z 406.157,A -85,B 0,C 180,E1 -25559.999,E2 -25559.999} C_VEL
LIN {X 0,Y 122.444,Z 406.231,A -85,B 0,C 180,E1 -25566.591,E2 -25566.591} C_VEL
LIN {X 0,Y 122.444,Z 406.228,A -85,B 0,C 180,E1 -25569.915,E2 -25569.915} C_VEL
LIN {X 0,Y 122.264,Z 406.246,A -85,B 0,C 180,E1 -25573.292,E2 -25573.292} C_VEL
LIN {X 0,Y 122.071,Z 406.275,A -85,B 0,C 180,E1 -25580.208,E2 -25580.208} C_VEL
LIN {X 0,Y 122.091,Z 406.447,A -85,B 0,C 180,E1 -25582.826,E2 -25582.826} C_VEL
LIN {X 0,Y 122.895,Z 408.97,A -85,B 0,C 180,E1 -25583.843,E2 -25583.843} C_VEL
LIN {X 0,Y 124.955,Z 411.227,A -85,B 0,C 180,E1 -25585.795,E2 -25585.795} C_VEL
LIN {X 0,Y 126.323,Z 412.2,A -85,B 0,C 180,E1 -25586.941,E2 -25586.941} C_VEL
LIN {X 0,Y 128.185,Z 415.391,A -85,B 0,C 180,E1 -25588.597,E2 -25588.597} C_VEL
LIN {X 0,Y 130.256,Z 417.446,A -85,B 0,C 180,E1 -25590.162,E2 -25590.162} C_VEL
LIN {X 0,Y 132.825,Z 421.102,A -85,B 0,C 180,E1 -25592.057,E2 -25592.057} C_VEL
LIN {X 0,Y 137.196,Z 427.362,A -85,B 0,C 180,E1 -25594.955,E2 -25594.955} C_VEL
LIN {X 0,Y 139.238,Z 430.853,A -85,B 0,C 180,E1 -25596.235,E2 -25596.235} C_VEL
LIN {X 0,Y 144.084,Z 440.981,A -85,B 0,C 180,E1 -25599.146,E2 -25599.146} C_VEL
LIN {X 0,Y 148.091,Z 450.839,A -85,B 0,C 180,E1 -25601.409,E2 -25601.409} C_VEL
LIN {X 0,Y 151.109,Z 459.911,A -85,B 0,C 180,E1 -25603.086,E2 -25603.086} C_VEL
LIN {X 0,Y 151.809,Z 474.069,A -85,B 0,C 180,E1 -25604.211,E2 -25604.211} C_VEL
LIN {X 0,Y 149.175,Z 512.179,A -85,B 0,C 180,E1 -25605.815,E2 -25605.815} C_VEL
LIN {X 0,Y 147.229,Z 525.806,A -85,B 0,C 180,E1 -25606.826,E2 -25606.826} C_VEL
LIN {X 0,Y 144.912,Z 537.589,A -85,B 0,C 180,E1 -25608.176,E2 -25608.176} C_VEL
LIN {X 0,Y 141.906,Z 548.893,A -85,B 0,C 180,E1 -25609.923,E2 -25609.923} C_VEL
LIN {X 0,Y 138.163,Z 560.594,A -85,B 0,C 180,E1 -25612.382,E2 -25612.382} C_VEL
LIN {X 0,Y 134.295,Z 571.119,A -85,B 0,C 180,E1 -25615.312,E2 -25615.312} C_VEL
LIN {X 0,Y 130.899,Z 579.728,A -85,B 0,C 180,E1 -25618.435,E2 -25618.435} C_VEL
LIN {X 0,Y 127.333,Z 587.986,A -85,B 0,C 180,E1 -25622.238,E2 -25622.238} C_VEL
LIN {X 0,Y 125.448,Z 592.994,A -85,B 0,C 180,E1 -25625.155,E2 -25625.155} C_VEL
LIN {X 0,Y 122.749,Z 599.697,A -85,B 0,C 180,E1 -25629.908,E2 -25629.908} C_VEL
LIN {X 0,Y 120.797,Z 605.028,A -85,B 0,C 180,E1 -25634.823,E2 -25634.823} C_VEL
LIN {X 0,Y 119.809,Z 609.174,A -85,B 0,C 180,E1 -25639.865,E2 -25639.865} C_VEL
LIN {X 0,Y 119.478,Z 611.328,A -85,B 0,C 180,E1 -25643.244,E2 -25643.244} C_VEL
LIN {X 0,Y 119.538,Z 613.667,A -85,B 0,C 180,E1 -25648.144,E2 -25648.144} C_VEL
LIN {X 0,Y 119.527,Z 614.751,A -85,B 0,C 180,E1 -25651.683,E2 -25651.683} C_VEL
LIN {X 0,Y 119.456,Z 615.531,A -85,B 0,C 180,E1 -25656.757,E2 -25656.757} C_VEL
LIN {X 0,Y 120.455,Z 615.159,A -85,B 0,C 180,E1 -25663.496,E2 -25663.496} C_VEL
LIN {X 0,Y 122.948,Z 613.25,A -85,B 0,C 180,E1 -25670.058,E2 -25670.058} C_VEL
LIN {X 0,Y 124.889,Z 611.665,A -85,B 0,C 180,E1 -25673.198,E2 -25673.198} C_VEL
LIN {X 0,Y 128.422,Z 608.518,A -85,B 0,C 180,E1 -25677.721,E2 -25677.721} C_VEL
LIN {X 0,Y 132.791,Z 604.17,A -85,B 0,C 180,E1 -25682.135,E2 -25682.135} C_VEL
LIN {X 0,Y 138.417,Z 597.991,A -85,B 0,C 180,E1 -25686.625,E2 -25686.625} C_VEL
LIN {X 0,Y 140.701,Z 595.366,A -85,B 0,C 180,E1 -25688.122,E2 -25688.122} C_VEL
LIN {X 0,Y 142.915,Z 592.141,A -85,B 0,C 180,E1 -25689.91,E2 -25689.91} C_VEL
LIN {X 0,Y 145.223,Z 586.546,A -85,B 0,C 180,E1 -25693.033,E2 -25693.033} C_VEL
LIN {X 0,Y 147.636,Z 580.451,A -85,B 0,C 180,E1 -25695.934,E2 -25695.934} C_VEL
LIN {X 0,Y 149.922,Z 576.362,A -85,B 0,C 180,E1 -25697.334,E2 -25697.334} C_VEL
LIN {X 0,Y 155.756,Z 566.866,A -85,B 0,C 180,E1 -25699.589,E2 -25699.589} C_VEL
LIN {X 0,Y 161.579,Z 555.671,A -85,B 0,C 180,E1 -25701.527,E2 -25701.527} C_VEL
LIN {X 0,Y 166.22,Z 544.727,A -85,B 0,C 180,E1 -25702.943,E2 -25702.943} C_VEL
LIN {X 0,Y 170.515,Z 531.948,A -85,B 0,C 180,E1 -25704.134,E2 -25704.134} C_VEL
LIN {X 0,Y 173.575,Z 519.117,A -85,B 0,C 180,E1 -25704.961,E2 -25704.961} C_VEL
LIN {X 0,Y 175.594,Z 505.197,A -85,B 0,C 180,E1 -25705.551,E2 -25705.551} C_VEL
LIN {X 0,Y 176.725,Z 491.754,A -85,B 0,C 180,E1 -25706.002,E2 -25706.002} C_VEL
LIN {X 0,Y 173.333,Z 482.191,A -85,B 0,C 180,E1 -25708.838,E2 -25708.838} C_VEL
LIN {X 0,Y 170.049,Z 474.101,A -85,B 0,C 180,E1 -25711.879,E2 -25711.879} C_VEL
LIN {X 0,Y 166.997,Z 467.323,A -85,B 0,C 180,E1 -25715.113,E2 -25715.113} C_VEL
LIN {X 0,Y 164.979,Z 463.122,A -85,B 0,C 180,E1 -25717.584,E2 -25717.584} C_VEL
LIN {X 0,Y 163.009,Z 459.119,A -85,B 0,C 180,E1 -25720.426,E2 -25720.426} C_VEL
LIN {X 0,Y 160.611,Z 455.062,A -85,B 0,C 180,E1 -25724.779,E2 -25724.779} C_VEL
LIN {X 0,Y 158.551,Z 452.128,A -85,B 0,C 180,E1 -25730.915,E2 -25730.915} C_VEL
LIN {X 0,Y 158.278,Z 450.198,A -85,B 0,C 180,E1 -25733.947,E2 -25733.947} C_VEL
LIN {X 0,Y 158.366,Z 450.245,A -85,B 0,C 180,E1 -25738.569,E2 -25738.569} C_VEL
LIN {X 0,Y 158.965,Z 452.847,A -85,B 0,C 180,E1 -25742.535,E2 -25742.535} C_VEL
LIN {X 0,Y 160.877,Z 455.225,A -85,B 0,C 180,E1 -25747.413,E2 -25747.413} C_VEL
LIN {X 0,Y 162.861,Z 458.742,A -85,B 0,C 180,E1 -25751.008,E2 -25751.008} C_VEL
LIN {X 0,Y 163.858,Z 460.226,A -85,B 0,C 180,E1 -25752.463,E2 -25752.463} C_VEL
LIN {X 0,Y 166.557,Z 464.555,A -85,B 0,C 180,E1 -25755.841,E2 -25755.841} C_VEL
LIN {X 0,Y 169.425,Z 469.29,A -85,B 0,C 180,E1 -25758.832,E2 -25758.832} C_VEL
LIN {X 0,Y 173.427,Z 476.588,A -85,B 0,C 180,E1 -25762.408,E2 -25762.408} C_VEL
LIN {X 0,Y 177.346,Z 484.444,A -85,B 0,C 180,E1 -25765.448,E2 -25765.448} C_VEL
LIN {X 0,Y 175.376,Z 504.05,A -85,B 0,C 180,E1 -25766.117,E2 -25766.117} C_VEL
LIN {X 0,Y 172.958,Z 517.221,A -85,B 0,C 180,E1 -25766.885,E2 -25766.885} C_VEL
LIN {X 0,Y 169.652,Z 529.652,A -85,B 0,C 180,E1 -25768.01,E2 -25768.01} C_VEL
LIN {X 0,Y 165.282,Z 541.404,A -85,B 0,C 180,E1 -25769.347,E2 -25769.347} C_VEL
LIN {X 0,Y 160.132,Z 552.735,A -85,B 0,C 180,E1 -25771.151,E2 -25771.151} C_VEL
LIN {X 0,Y 154.748,Z 562.855,A -85,B 0,C 180,E1 -25773.425,E2 -25773.425} C_VEL
LIN {X 0,Y 148.23,Z 572.816,A -85,B 0,C 180,E1 -25776.293,E2 -25776.293} C_VEL
LIN {X 0,Y 142.544,Z 580.306,A -85,B 0,C 180,E1 -25779.169,E2 -25779.169} C_VEL
LIN {X 0,Y 136.491,Z 587.361,A -85,B 0,C 180,E1 -25782.8,E2 -25782.8} C_VEL
LIN {X 0,Y 131.759,Z 592.188,A -85,B 0,C 180,E1 -25786.1,E2 -25786.1} C_VEL
LIN {X 0,Y 126.672,Z 596.837,A -85,B 0,C 180,E1 -25790.355,E2 -25790.355} C_VEL
LIN {X 0,Y 122.251,Z 600.345,A -85,B 0,C 180,E1 -25794.91,E2 -25794.91} C_VEL
